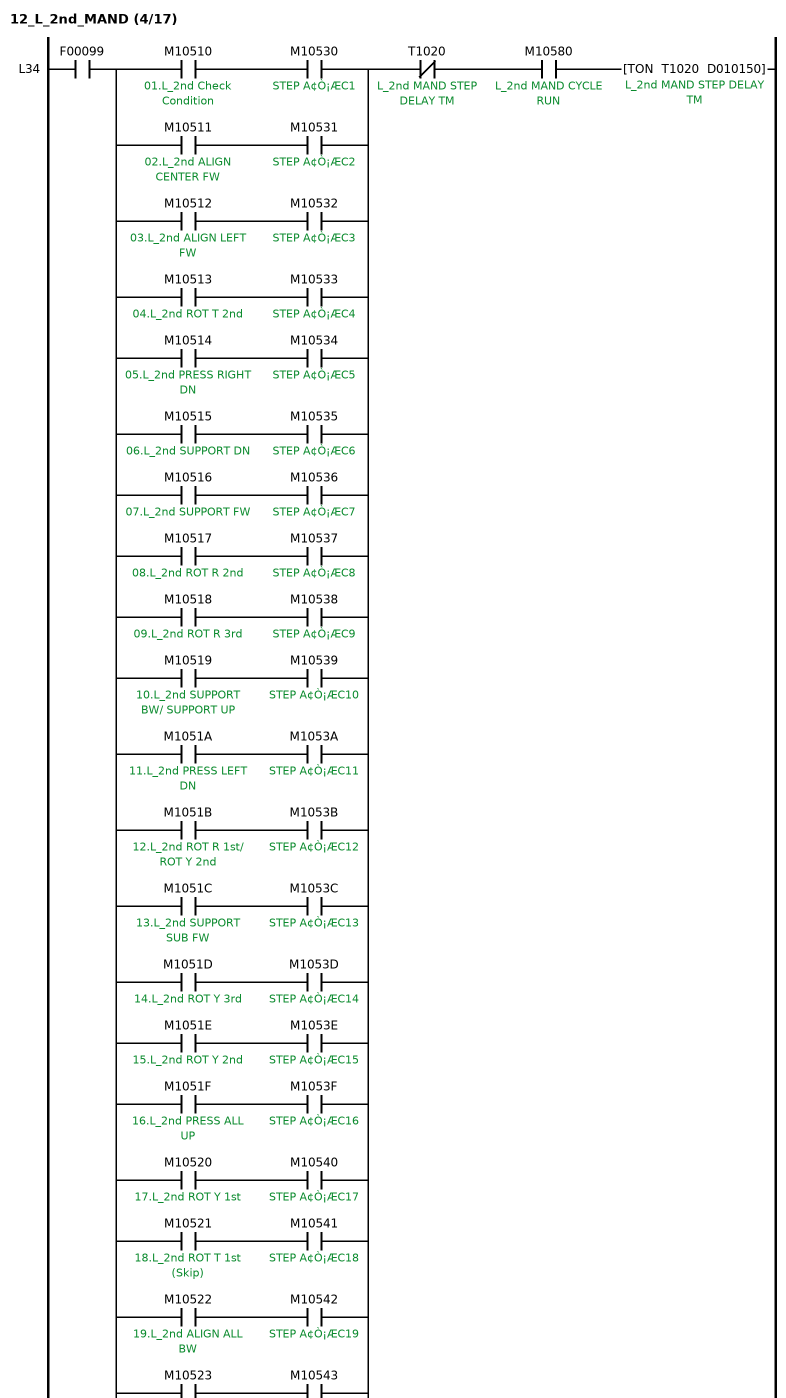
[picture p72: 12_L_2nd_MAND rungs L34-L34]

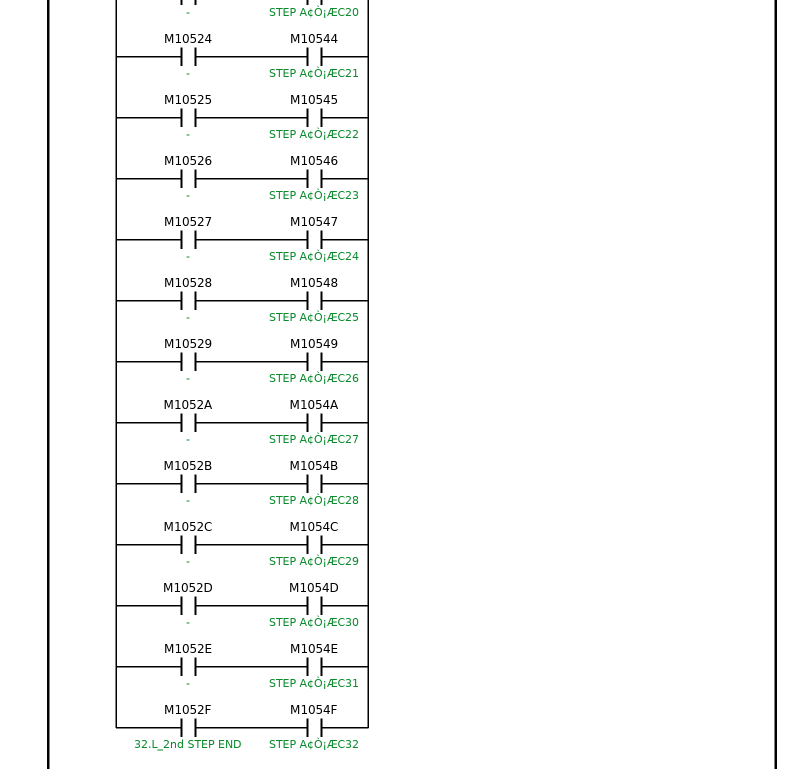
; L34
LOAD      F00099
LOAD      M10510	// 01.L_2nd Check Condition
AND       M10530	// STEP A¢Ò¡ÆC1
LOAD      M10511	// 02.L_2nd ALIGN CENTER FW
AND       M10531	// STEP A¢Ò¡ÆC2
OR LOAD
LOAD      M10512	// 03.L_2nd ALIGN LEFT FW
AND       M10532	// STEP A¢Ò¡ÆC3
OR LOAD
LOAD      M10513	// 04.L_2nd ROT T 2nd
AND       M10533	// STEP A¢Ò¡ÆC4
OR LOAD
LOAD      M10514	// 05.L_2nd PRESS RIGHT DN
AND       M10534	// STEP A¢Ò¡ÆC5
OR LOAD
LOAD      M10515	// 06.L_2nd SUPPORT DN
AND       M10535	// STEP A¢Ò¡ÆC6
OR LOAD
LOAD      M10516	// 07.L_2nd SUPPORT FW
AND       M10536	// STEP A¢Ò¡ÆC7
OR LOAD
LOAD      M10517	// 08.L_2nd ROT R 2nd
AND       M10537	// STEP A¢Ò¡ÆC8
OR LOAD
LOAD      M10518	// 09.L_2nd ROT R 3rd
AND       M10538	// STEP A¢Ò¡ÆC9
OR LOAD
LOAD      M10519	// 10.L_2nd SUPPORT BW/ SUPPORT UP
AND       M10539	// STEP A¢Ò¡ÆC10
OR LOAD
LOAD      M1051A	// 11.L_2nd PRESS LEFT DN
AND       M1053A	// STEP A¢Ò¡ÆC11
OR LOAD
LOAD      M1051B	// 12.L_2nd ROT R 1st/ ROT Y 2nd
AND       M1053B	// STEP A¢Ò¡ÆC12
OR LOAD
LOAD      M1051C	// 13.L_2nd SUPPORT SUB FW
AND       M1053C	// STEP A¢Ò¡ÆC13
OR LOAD
LOAD      M1051D	// 14.L_2nd ROT Y 3rd
AND       M1053D	// STEP A¢Ò¡ÆC14
OR LOAD
LOAD      M1051E	// 15.L_2nd ROT Y 2nd
AND       M1053E	// STEP A¢Ò¡ÆC15
OR LOAD
LOAD      M1051F	// 16.L_2nd PRESS ALL UP
AND       M1053F	// STEP A¢Ò¡ÆC16
OR LOAD
LOAD      M10520	// 17.L_2nd ROT Y 1st
AND       M10540	// STEP A¢Ò¡ÆC17
OR LOAD
LOAD      M10521	// 18.L_2nd ROT T 1st (Skip)
AND       M10541	// STEP A¢Ò¡ÆC18
OR LOAD
LOAD      M10522	// 19.L_2nd ALIGN ALL BW
AND       M10542	// STEP A¢Ò¡ÆC19
OR LOAD
LOAD      M10523	// -
AND       M10543	// STEP A¢Ò¡ÆC20
OR LOAD
LOAD      M10524	// -
AND       M10544	// STEP A¢Ò¡ÆC21
OR LOAD
LOAD      M10525	// -
AND       M10545	// STEP A¢Ò¡ÆC22
OR LOAD
LOAD      M10526	// -
AND       M10546	// STEP A¢Ò¡ÆC23
OR LOAD
LOAD      M10527	// -
AND       M10547	// STEP A¢Ò¡ÆC24
OR LOAD
LOAD      M10528	// -
AND       M10548	// STEP A¢Ò¡ÆC25
OR LOAD
LOAD      M10529	// -
AND       M10549	// STEP A¢Ò¡ÆC26
OR LOAD
LOAD      M1052A	// -
AND       M1054A	// STEP A¢Ò¡ÆC27
OR LOAD
LOAD      M1052B	// -
AND       M1054B	// STEP A¢Ò¡ÆC28
OR LOAD
LOAD      M1052C	// -
AND       M1054C	// STEP A¢Ò¡ÆC29
OR LOAD
LOAD      M1052D	// -
AND       M1054D	// STEP A¢Ò¡ÆC30
OR LOAD
LOAD      M1052E	// -
AND       M1054E	// STEP A¢Ò¡ÆC31
OR LOAD
LOAD      M1052F	// 32.L_2nd STEP END
AND       M1054F	// STEP A¢Ò¡ÆC32
OR LOAD
AND LOAD
AND NOT   T1020	// L_2nd MAND STEP DELAY TM
AND       M10580	// L_2nd MAND CYCLE RUN
TON       T1020 D010150	// L_2nd MAND STEP DELAY TM

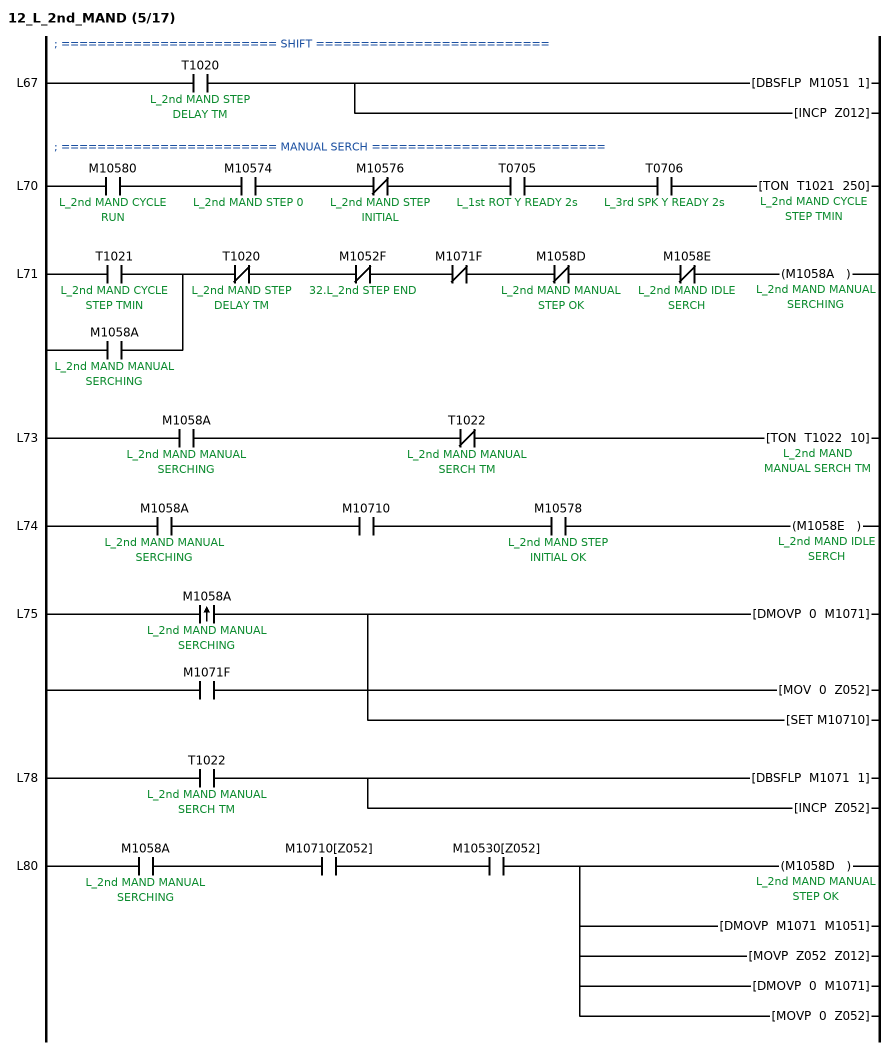
// ======================== SHIFT ==========================
; L67
LOAD      T1020	// L_2nd MAND STEP DELAY TM
DBSFLP    M1051 1
INCP      Z012
// ======================== MANUAL SERCH ==========================
; L70
LOAD      M10580	// L_2nd MAND CYCLE RUN
AND       M10574	// L_2nd MAND STEP 0
AND NOT   M10576	// L_2nd MAND STEP INITIAL
AND       T0705	// L_1st ROT Y READY 2s
AND       T0706	// L_3rd SPK Y READY 2s
TON       T1021 250	// L_2nd MAND CYCLE STEP TMIN
; L71
LOAD      T1021	// L_2nd MAND CYCLE STEP TMIN
OR        M1058A	// L_2nd MAND MANUAL SERCHING
AND NOT   T1020	// L_2nd MAND STEP DELAY TM
AND NOT   M1052F	// 32.L_2nd STEP END
AND NOT   M1071F
AND NOT   M1058D	// L_2nd MAND MANUAL STEP OK
AND NOT   M1058E	// L_2nd MAND IDLE SERCH
OUT       M1058A	// L_2nd MAND MANUAL SERCHING
; L73
LOAD      M1058A	// L_2nd MAND MANUAL SERCHING
AND NOT   T1022	// L_2nd MAND MANUAL SERCH TM
TON       T1022 10	// L_2nd MAND MANUAL SERCH TM
; L74
LOAD      M1058A	// L_2nd MAND MANUAL SERCHING
AND       M10710
AND       M10578	// L_2nd MAND STEP INITIAL OK
OUT       M1058E	// L_2nd MAND IDLE SERCH
; L75
LOADP     M1058A	// L_2nd MAND MANUAL SERCHING
OR        M1071F
DMOVP     0 M1071
MOV       0 Z052
SET       M10710
; L78
LOAD      T1022	// L_2nd MAND MANUAL SERCH TM
DBSFLP    M1071 1
INCP      Z052
; L80
LOAD      M1058A	// L_2nd MAND MANUAL SERCHING
AND       M10710[Z052]
AND       M10530[Z052]
OUT       M1058D	// L_2nd MAND MANUAL STEP OK
DMOVP     M1071 M1051
MOVP      Z052 Z012
DMOVP     0 M1071
MOVP      0 Z052

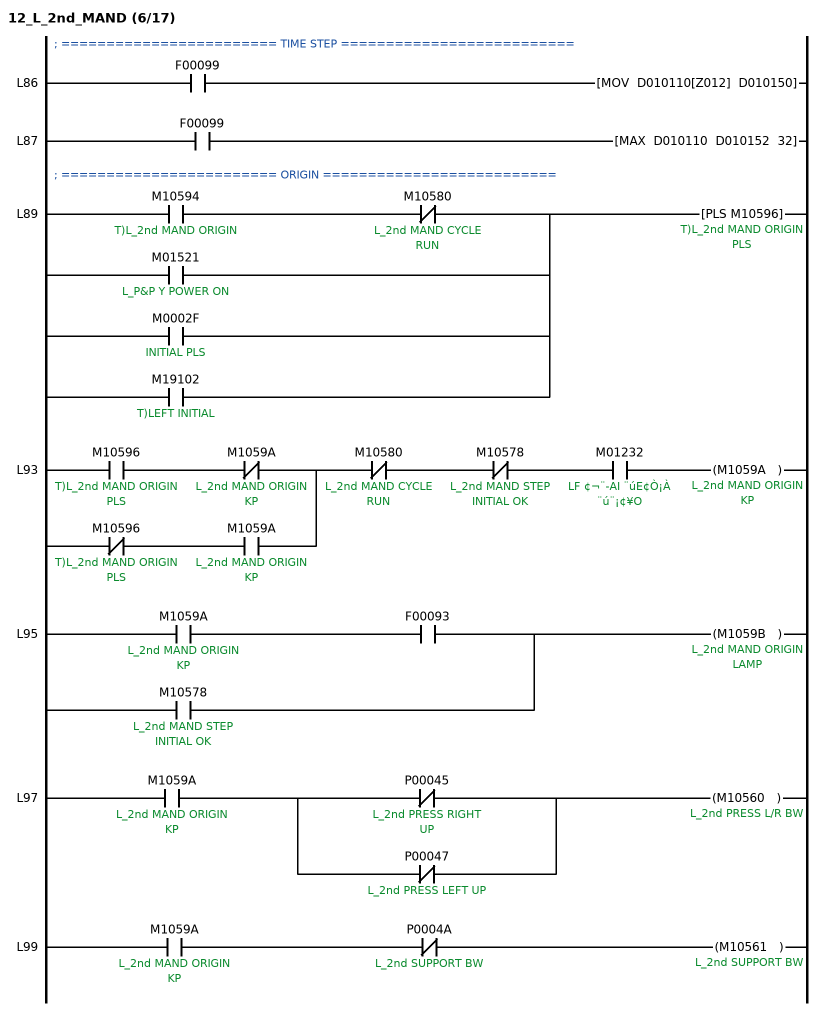
// ======================== TIME STEP ==========================
; L86
LOAD      F00099
MOV       D010110[Z012] D010150
; L87
LOAD      F00099
MAX       D010110 D010152 32
// ======================== ORIGIN ==========================
; L89
LOAD      M10594	// T)L_2nd MAND ORIGIN
AND NOT   M10580	// L_2nd MAND CYCLE RUN
OR        M01521	// L_P&P Y POWER ON
OR        M0002F	// INITIAL PLS
OR        M19102	// T)LEFT INITIAL
OUTP      M10596	// T)L_2nd MAND ORIGIN PLS
; L93
LOAD      M10596	// T)L_2nd MAND ORIGIN PLS
AND NOT   M1059A	// L_2nd MAND ORIGIN KP
LOAD NOT  M10596	// T)L_2nd MAND ORIGIN PLS
AND       M1059A	// L_2nd MAND ORIGIN KP
OR LOAD
AND NOT   M10580	// L_2nd MAND CYCLE RUN
AND NOT   M10578	// L_2nd MAND STEP INITIAL OK
AND       M01232	// LF ¢¬¨­AI ¨úE¢Ò¡À ¨ú¨¡¢¥O
OUT       M1059A	// L_2nd MAND ORIGIN KP
; L95
LOAD      M1059A	// L_2nd MAND ORIGIN KP
AND       F00093
OR        M10578	// L_2nd MAND STEP INITIAL OK
OUT       M1059B	// L_2nd MAND ORIGIN LAMP
; L97
LOAD      M1059A	// L_2nd MAND ORIGIN KP
LOAD NOT  P00045	// L_2nd PRESS RIGHT UP
OR NOT    P00047	// L_2nd PRESS LEFT UP
AND LOAD
OUT       M10560	// L_2nd PRESS L/R BW
; L99
LOAD      M1059A	// L_2nd MAND ORIGIN KP
AND NOT   P0004A	// L_2nd SUPPORT BW
OUT       M10561	// L_2nd SUPPORT BW

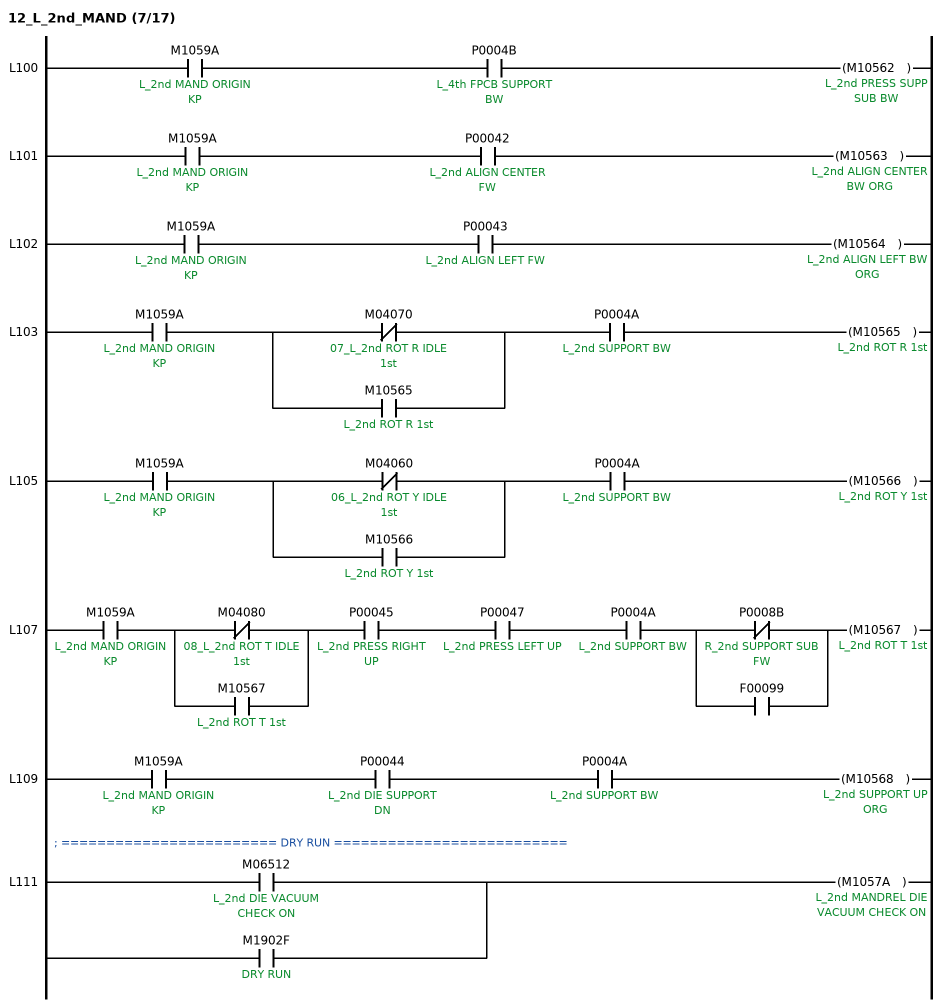
; L100
LOAD      M1059A	// L_2nd MAND ORIGIN KP
AND       P0004B	// L_4th FPCB SUPPORT BW
OUT       M10562	// L_2nd PRESS SUPP SUB BW
; L101
LOAD      M1059A	// L_2nd MAND ORIGIN KP
AND       P00042	// L_2nd ALIGN CENTER FW
OUT       M10563	// L_2nd ALIGN CENTER BW ORG
; L102
LOAD      M1059A	// L_2nd MAND ORIGIN KP
AND       P00043	// L_2nd ALIGN LEFT FW
OUT       M10564	// L_2nd ALIGN LEFT BW ORG
; L103
LOAD      M1059A	// L_2nd MAND ORIGIN KP
LOAD NOT  M04070	// 07_L_2nd ROT R IDLE 1st
OR        M10565	// L_2nd ROT R 1st
AND LOAD
AND       P0004A	// L_2nd SUPPORT BW
OUT       M10565	// L_2nd ROT R 1st
; L105
LOAD      M1059A	// L_2nd MAND ORIGIN KP
LOAD NOT  M04060	// 06_L_2nd ROT Y IDLE 1st
OR        M10566	// L_2nd ROT Y 1st
AND LOAD
AND       P0004A	// L_2nd SUPPORT BW
OUT       M10566	// L_2nd ROT Y 1st
; L107
LOAD      M1059A	// L_2nd MAND ORIGIN KP
LOAD NOT  M04080	// 08_L_2nd ROT T IDLE 1st
OR        M10567	// L_2nd ROT T 1st
AND LOAD
AND       P00045	// L_2nd PRESS RIGHT UP
AND       P00047	// L_2nd PRESS LEFT UP
AND       P0004A	// L_2nd SUPPORT BW
LOAD NOT  P0008B	// R_2nd SUPPORT SUB FW
OR        F00099
AND LOAD
OUT       M10567	// L_2nd ROT T 1st
; L109
LOAD      M1059A	// L_2nd MAND ORIGIN KP
AND       P00044	// L_2nd DIE SUPPORT DN
AND       P0004A	// L_2nd SUPPORT BW
OUT       M10568	// L_2nd SUPPORT UP ORG
// ======================== DRY RUN ==========================
; L111
LOAD      M06512	// L_2nd DIE VACUUM CHECK ON
OR        M1902F	// DRY RUN
OUT       M1057A	// L_2nd MANDREL DIE VACUUM CHECK ON

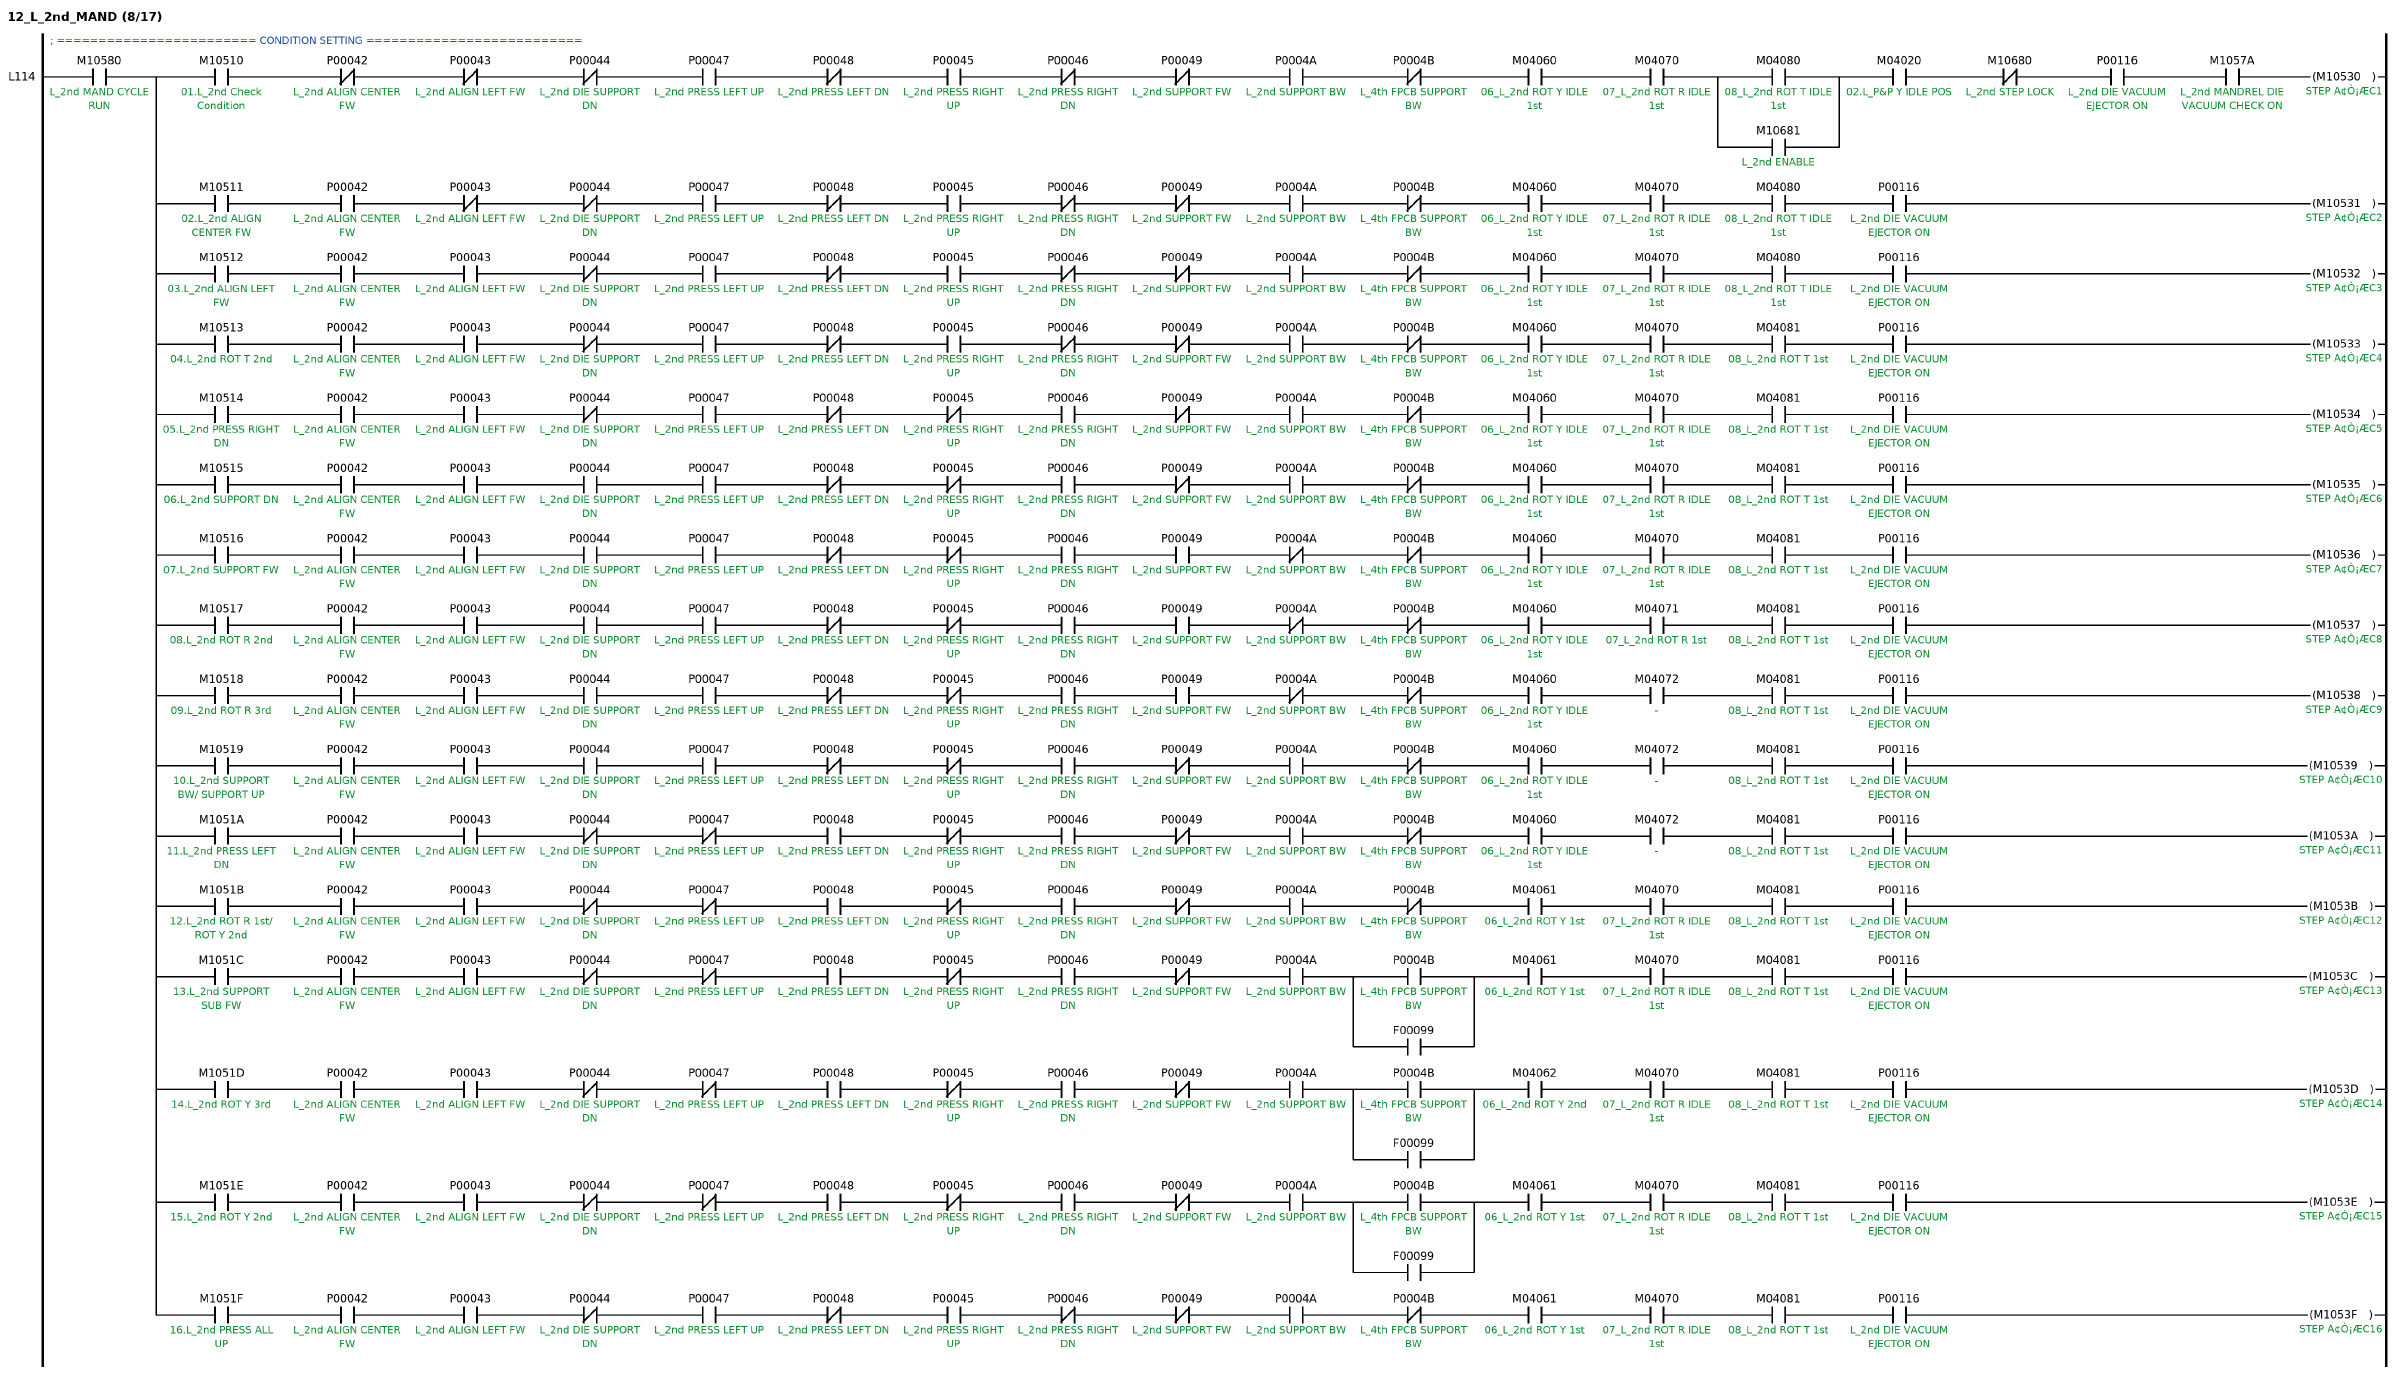
// ======================== CONDITION SETTING ==========================
; L114
LOAD      M10580	// L_2nd MAND CYCLE RUN
MPUSH
AND       M10510	// 01.L_2nd Check Condition
AND NOT   P00042	// L_2nd ALIGN CENTER FW
AND NOT   P00043	// L_2nd ALIGN LEFT FW
AND NOT   P00044	// L_2nd DIE SUPPORT DN
AND       P00047	// L_2nd PRESS LEFT UP
AND NOT   P00048	// L_2nd PRESS LEFT DN
AND       P00045	// L_2nd PRESS RIGHT UP
AND NOT   P00046	// L_2nd PRESS RIGHT DN
AND NOT   P00049	// L_2nd SUPPORT FW
AND       P0004A	// L_2nd SUPPORT BW
AND NOT   P0004B	// L_4th FPCB SUPPORT BW
AND       M04060	// 06_L_2nd ROT Y IDLE 1st
AND       M04070	// 07_L_2nd ROT R IDLE 1st
LOAD      M04080	// 08_L_2nd ROT T IDLE 1st
OR        M10681	// L_2nd ENABLE
AND LOAD
AND       M04020	// 02.L_P&P Y IDLE POS
AND NOT   M10680	// L_2nd STEP LOCK
AND       P00116	// L_2nd DIE VACUUM EJECTOR ON
AND       M1057A	// L_2nd MANDREL DIE VACUUM CHECK ON
OUT       M10530	// STEP A¢Ò¡ÆC1
MLOAD
AND       M10511	// 02.L_2nd ALIGN CENTER FW
AND       P00042	// L_2nd ALIGN CENTER FW
AND NOT   P00043	// L_2nd ALIGN LEFT FW
AND NOT   P00044	// L_2nd DIE SUPPORT DN
AND       P00047	// L_2nd PRESS LEFT UP
AND NOT   P00048	// L_2nd PRESS LEFT DN
AND       P00045	// L_2nd PRESS RIGHT UP
AND NOT   P00046	// L_2nd PRESS RIGHT DN
AND NOT   P00049	// L_2nd SUPPORT FW
AND       P0004A	// L_2nd SUPPORT BW
AND NOT   P0004B	// L_4th FPCB SUPPORT BW
AND       M04060	// 06_L_2nd ROT Y IDLE 1st
AND       M04070	// 07_L_2nd ROT R IDLE 1st
AND       M04080	// 08_L_2nd ROT T IDLE 1st
AND       P00116	// L_2nd DIE VACUUM EJECTOR ON
OUT       M10531	// STEP A¢Ò¡ÆC2
MLOAD
AND       M10512	// 03.L_2nd ALIGN LEFT FW
AND       P00042	// L_2nd ALIGN CENTER FW
AND       P00043	// L_2nd ALIGN LEFT FW
AND NOT   P00044	// L_2nd DIE SUPPORT DN
AND       P00047	// L_2nd PRESS LEFT UP
AND NOT   P00048	// L_2nd PRESS LEFT DN
AND       P00045	// L_2nd PRESS RIGHT UP
AND NOT   P00046	// L_2nd PRESS RIGHT DN
AND NOT   P00049	// L_2nd SUPPORT FW
AND       P0004A	// L_2nd SUPPORT BW
AND NOT   P0004B	// L_4th FPCB SUPPORT BW
AND       M04060	// 06_L_2nd ROT Y IDLE 1st
AND       M04070	// 07_L_2nd ROT R IDLE 1st
AND       M04080	// 08_L_2nd ROT T IDLE 1st
AND       P00116	// L_2nd DIE VACUUM EJECTOR ON
OUT       M10532	// STEP A¢Ò¡ÆC3
MLOAD
AND       M10513	// 04.L_2nd ROT T 2nd
AND       P00042	// L_2nd ALIGN CENTER FW
AND       P00043	// L_2nd ALIGN LEFT FW
AND NOT   P00044	// L_2nd DIE SUPPORT DN
AND       P00047	// L_2nd PRESS LEFT UP
AND NOT   P00048	// L_2nd PRESS LEFT DN
AND       P00045	// L_2nd PRESS RIGHT UP
AND NOT   P00046	// L_2nd PRESS RIGHT DN
AND NOT   P00049	// L_2nd SUPPORT FW
AND       P0004A	// L_2nd SUPPORT BW
AND NOT   P0004B	// L_4th FPCB SUPPORT BW
AND       M04060	// 06_L_2nd ROT Y IDLE 1st
AND       M04070	// 07_L_2nd ROT R IDLE 1st
AND       M04081	// 08_L_2nd ROT T 1st
AND       P00116	// L_2nd DIE VACUUM EJECTOR ON
OUT       M10533	// STEP A¢Ò¡ÆC4
MLOAD
AND       M10514	// 05.L_2nd PRESS RIGHT DN
AND       P00042	// L_2nd ALIGN CENTER FW
AND       P00043	// L_2nd ALIGN LEFT FW
AND NOT   P00044	// L_2nd DIE SUPPORT DN
AND       P00047	// L_2nd PRESS LEFT UP
AND NOT   P00048	// L_2nd PRESS LEFT DN
AND NOT   P00045	// L_2nd PRESS RIGHT UP
AND       P00046	// L_2nd PRESS RIGHT DN
AND NOT   P00049	// L_2nd SUPPORT FW
AND       P0004A	// L_2nd SUPPORT BW
AND NOT   P0004B	// L_4th FPCB SUPPORT BW
AND       M04060	// 06_L_2nd ROT Y IDLE 1st
AND       M04070	// 07_L_2nd ROT R IDLE 1st
AND       M04081	// 08_L_2nd ROT T 1st
AND       P00116	// L_2nd DIE VACUUM EJECTOR ON
OUT       M10534	// STEP A¢Ò¡ÆC5
MLOAD
AND       M10515	// 06.L_2nd SUPPORT DN
AND       P00042	// L_2nd ALIGN CENTER FW
AND       P00043	// L_2nd ALIGN LEFT FW
AND       P00044	// L_2nd DIE SUPPORT DN
AND       P00047	// L_2nd PRESS LEFT UP
AND NOT   P00048	// L_2nd PRESS LEFT DN
AND NOT   P00045	// L_2nd PRESS RIGHT UP
AND       P00046	// L_2nd PRESS RIGHT DN
AND NOT   P00049	// L_2nd SUPPORT FW
AND       P0004A	// L_2nd SUPPORT BW
AND NOT   P0004B	// L_4th FPCB SUPPORT BW
AND       M04060	// 06_L_2nd ROT Y IDLE 1st
AND       M04070	// 07_L_2nd ROT R IDLE 1st
AND       M04081	// 08_L_2nd ROT T 1st
AND       P00116	// L_2nd DIE VACUUM EJECTOR ON
OUT       M10535	// STEP A¢Ò¡ÆC6
MLOAD
AND       M10516	// 07.L_2nd SUPPORT FW
AND       P00042	// L_2nd ALIGN CENTER FW
AND       P00043	// L_2nd ALIGN LEFT FW
AND       P00044	// L_2nd DIE SUPPORT DN
AND       P00047	// L_2nd PRESS LEFT UP
AND NOT   P00048	// L_2nd PRESS LEFT DN
AND NOT   P00045	// L_2nd PRESS RIGHT UP
AND       P00046	// L_2nd PRESS RIGHT DN
AND       P00049	// L_2nd SUPPORT FW
AND NOT   P0004A	// L_2nd SUPPORT BW
AND NOT   P0004B	// L_4th FPCB SUPPORT BW
AND       M04060	// 06_L_2nd ROT Y IDLE 1st
AND       M04070	// 07_L_2nd ROT R IDLE 1st
AND       M04081	// 08_L_2nd ROT T 1st
AND       P00116	// L_2nd DIE VACUUM EJECTOR ON
OUT       M10536	// STEP A¢Ò¡ÆC7
MLOAD
AND       M10517	// 08.L_2nd ROT R 2nd
AND       P00042	// L_2nd ALIGN CENTER FW
AND       P00043	// L_2nd ALIGN LEFT FW
AND       P00044	// L_2nd DIE SUPPORT DN
AND       P00047	// L_2nd PRESS LEFT UP
AND NOT   P00048	// L_2nd PRESS LEFT DN
AND NOT   P00045	// L_2nd PRESS RIGHT UP
AND       P00046	// L_2nd PRESS RIGHT DN
AND       P00049	// L_2nd SUPPORT FW
AND NOT   P0004A	// L_2nd SUPPORT BW
AND NOT   P0004B	// L_4th FPCB SUPPORT BW
AND       M04060	// 06_L_2nd ROT Y IDLE 1st
AND       M04071	// 07_L_2nd ROT R 1st
AND       M04081	// 08_L_2nd ROT T 1st
AND       P00116	// L_2nd DIE VACUUM EJECTOR ON
OUT       M10537	// STEP A¢Ò¡ÆC8
MLOAD
AND       M10518	// 09.L_2nd ROT R 3rd
AND       P00042	// L_2nd ALIGN CENTER FW
AND       P00043	// L_2nd ALIGN LEFT FW
AND       P00044	// L_2nd DIE SUPPORT DN
AND       P00047	// L_2nd PRESS LEFT UP
AND NOT   P00048	// L_2nd PRESS LEFT DN
AND NOT   P00045	// L_2nd PRESS RIGHT UP
AND       P00046	// L_2nd PRESS RIGHT DN
AND       P00049	// L_2nd SUPPORT FW
AND NOT   P0004A	// L_2nd SUPPORT BW
AND NOT   P0004B	// L_4th FPCB SUPPORT BW
AND       M04060	// 06_L_2nd ROT Y IDLE 1st
AND       M04072	// -
AND       M04081	// 08_L_2nd ROT T 1st
AND       P00116	// L_2nd DIE VACUUM EJECTOR ON
OUT       M10538	// STEP A¢Ò¡ÆC9
MLOAD
AND       M10519	// 10.L_2nd SUPPORT BW/ SUPPORT UP
AND       P00042	// L_2nd ALIGN CENTER FW
AND       P00043	// L_2nd ALIGN LEFT FW
AND       P00044	// L_2nd DIE SUPPORT DN
AND       P00047	// L_2nd PRESS LEFT UP
AND NOT   P00048	// L_2nd PRESS LEFT DN
AND NOT   P00045	// L_2nd PRESS RIGHT UP
AND       P00046	// L_2nd PRESS RIGHT DN
AND NOT   P00049	// L_2nd SUPPORT FW
AND       P0004A	// L_2nd SUPPORT BW
AND NOT   P0004B	// L_4th FPCB SUPPORT BW
AND       M04060	// 06_L_2nd ROT Y IDLE 1st
AND       M04072	// -
AND       M04081	// 08_L_2nd ROT T 1st
AND       P00116	// L_2nd DIE VACUUM EJECTOR ON
OUT       M10539	// STEP A¢Ò¡ÆC10
MLOAD
AND       M1051A	// 11.L_2nd PRESS LEFT DN
AND       P00042	// L_2nd ALIGN CENTER FW
AND       P00043	// L_2nd ALIGN LEFT FW
AND NOT   P00044	// L_2nd DIE SUPPORT DN
AND NOT   P00047	// L_2nd PRESS LEFT UP
AND       P00048	// L_2nd PRESS LEFT DN
AND NOT   P00045	// L_2nd PRESS RIGHT UP
AND       P00046	// L_2nd PRESS RIGHT DN
AND NOT   P00049	// L_2nd SUPPORT FW
AND       P0004A	// L_2nd SUPPORT BW
AND NOT   P0004B	// L_4th FPCB SUPPORT BW
AND       M04060	// 06_L_2nd ROT Y IDLE 1st
AND       M04072	// -
AND       M04081	// 08_L_2nd ROT T 1st
AND       P00116	// L_2nd DIE VACUUM EJECTOR ON
OUT       M1053A	// STEP A¢Ò¡ÆC11
MLOAD
AND       M1051B	// 12.L_2nd ROT R 1st/ ROT Y 2nd
AND       P00042	// L_2nd ALIGN CENTER FW
AND       P00043	// L_2nd ALIGN LEFT FW
AND NOT   P00044	// L_2nd DIE SUPPORT DN
AND NOT   P00047	// L_2nd PRESS LEFT UP
AND       P00048	// L_2nd PRESS LEFT DN
AND NOT   P00045	// L_2nd PRESS RIGHT UP
AND       P00046	// L_2nd PRESS RIGHT DN
AND NOT   P00049	// L_2nd SUPPORT FW
AND       P0004A	// L_2nd SUPPORT BW
AND NOT   P0004B	// L_4th FPCB SUPPORT BW
AND       M04061	// 06_L_2nd ROT Y 1st
AND       M04070	// 07_L_2nd ROT R IDLE 1st
AND       M04081	// 08_L_2nd ROT T 1st
AND       P00116	// L_2nd DIE VACUUM EJECTOR ON
OUT       M1053B	// STEP A¢Ò¡ÆC12
MLOAD
AND       M1051C	// 13.L_2nd SUPPORT SUB FW
AND       P00042	// L_2nd ALIGN CENTER FW
AND       P00043	// L_2nd ALIGN LEFT FW
AND NOT   P00044	// L_2nd DIE SUPPORT DN
AND NOT   P00047	// L_2nd PRESS LEFT UP
AND       P00048	// L_2nd PRESS LEFT DN
AND NOT   P00045	// L_2nd PRESS RIGHT UP
AND       P00046	// L_2nd PRESS RIGHT DN
AND NOT   P00049	// L_2nd SUPPORT FW
AND       P0004A	// L_2nd SUPPORT BW
LOAD      P0004B	// L_4th FPCB SUPPORT BW
OR        F00099
AND LOAD
AND       M04061	// 06_L_2nd ROT Y 1st
AND       M04070	// 07_L_2nd ROT R IDLE 1st
AND       M04081	// 08_L_2nd ROT T 1st
AND       P00116	// L_2nd DIE VACUUM EJECTOR ON
OUT       M1053C	// STEP A¢Ò¡ÆC13
MLOAD
AND       M1051D	// 14.L_2nd ROT Y 3rd
AND       P00042	// L_2nd ALIGN CENTER FW
AND       P00043	// L_2nd ALIGN LEFT FW
AND NOT   P00044	// L_2nd DIE SUPPORT DN
AND NOT   P00047	// L_2nd PRESS LEFT UP
AND       P00048	// L_2nd PRESS LEFT DN
AND NOT   P00045	// L_2nd PRESS RIGHT UP
AND       P00046	// L_2nd PRESS RIGHT DN
AND NOT   P00049	// L_2nd SUPPORT FW
AND       P0004A	// L_2nd SUPPORT BW
LOAD      P0004B	// L_4th FPCB SUPPORT BW
OR        F00099
AND LOAD
AND       M04062	// 06_L_2nd ROT Y 2nd
AND       M04070	// 07_L_2nd ROT R IDLE 1st
AND       M04081	// 08_L_2nd ROT T 1st
AND       P00116	// L_2nd DIE VACUUM EJECTOR ON
OUT       M1053D	// STEP A¢Ò¡ÆC14
MLOAD
AND       M1051E	// 15.L_2nd ROT Y 2nd
AND       P00042	// L_2nd ALIGN CENTER FW
AND       P00043	// L_2nd ALIGN LEFT FW
AND NOT   P00044	// L_2nd DIE SUPPORT DN
AND NOT   P00047	// L_2nd PRESS LEFT UP
AND       P00048	// L_2nd PRESS LEFT DN
AND NOT   P00045	// L_2nd PRESS RIGHT UP
AND       P00046	// L_2nd PRESS RIGHT DN
AND NOT   P00049	// L_2nd SUPPORT FW
AND       P0004A	// L_2nd SUPPORT BW
LOAD      P0004B	// L_4th FPCB SUPPORT BW
OR        F00099
AND LOAD
AND       M04061	// 06_L_2nd ROT Y 1st
AND       M04070	// 07_L_2nd ROT R IDLE 1st
AND       M04081	// 08_L_2nd ROT T 1st
AND       P00116	// L_2nd DIE VACUUM EJECTOR ON
OUT       M1053E	// STEP A¢Ò¡ÆC15
MPOP
AND       M1051F	// 16.L_2nd PRESS ALL UP
AND       P00042	// L_2nd ALIGN CENTER FW
AND       P00043	// L_2nd ALIGN LEFT FW
AND NOT   P00044	// L_2nd DIE SUPPORT DN
AND       P00047	// L_2nd PRESS LEFT UP
AND NOT   P00048	// L_2nd PRESS LEFT DN
AND       P00045	// L_2nd PRESS RIGHT UP
AND NOT   P00046	// L_2nd PRESS RIGHT DN
AND NOT   P00049	// L_2nd SUPPORT FW
AND       P0004A	// L_2nd SUPPORT BW
AND NOT   P0004B	// L_4th FPCB SUPPORT BW
AND       M04061	// 06_L_2nd ROT Y 1st
AND       M04070	// 07_L_2nd ROT R IDLE 1st
AND       M04081	// 08_L_2nd ROT T 1st
AND       P00116	// L_2nd DIE VACUUM EJECTOR ON
OUT       M1053F	// STEP A¢Ò¡ÆC16

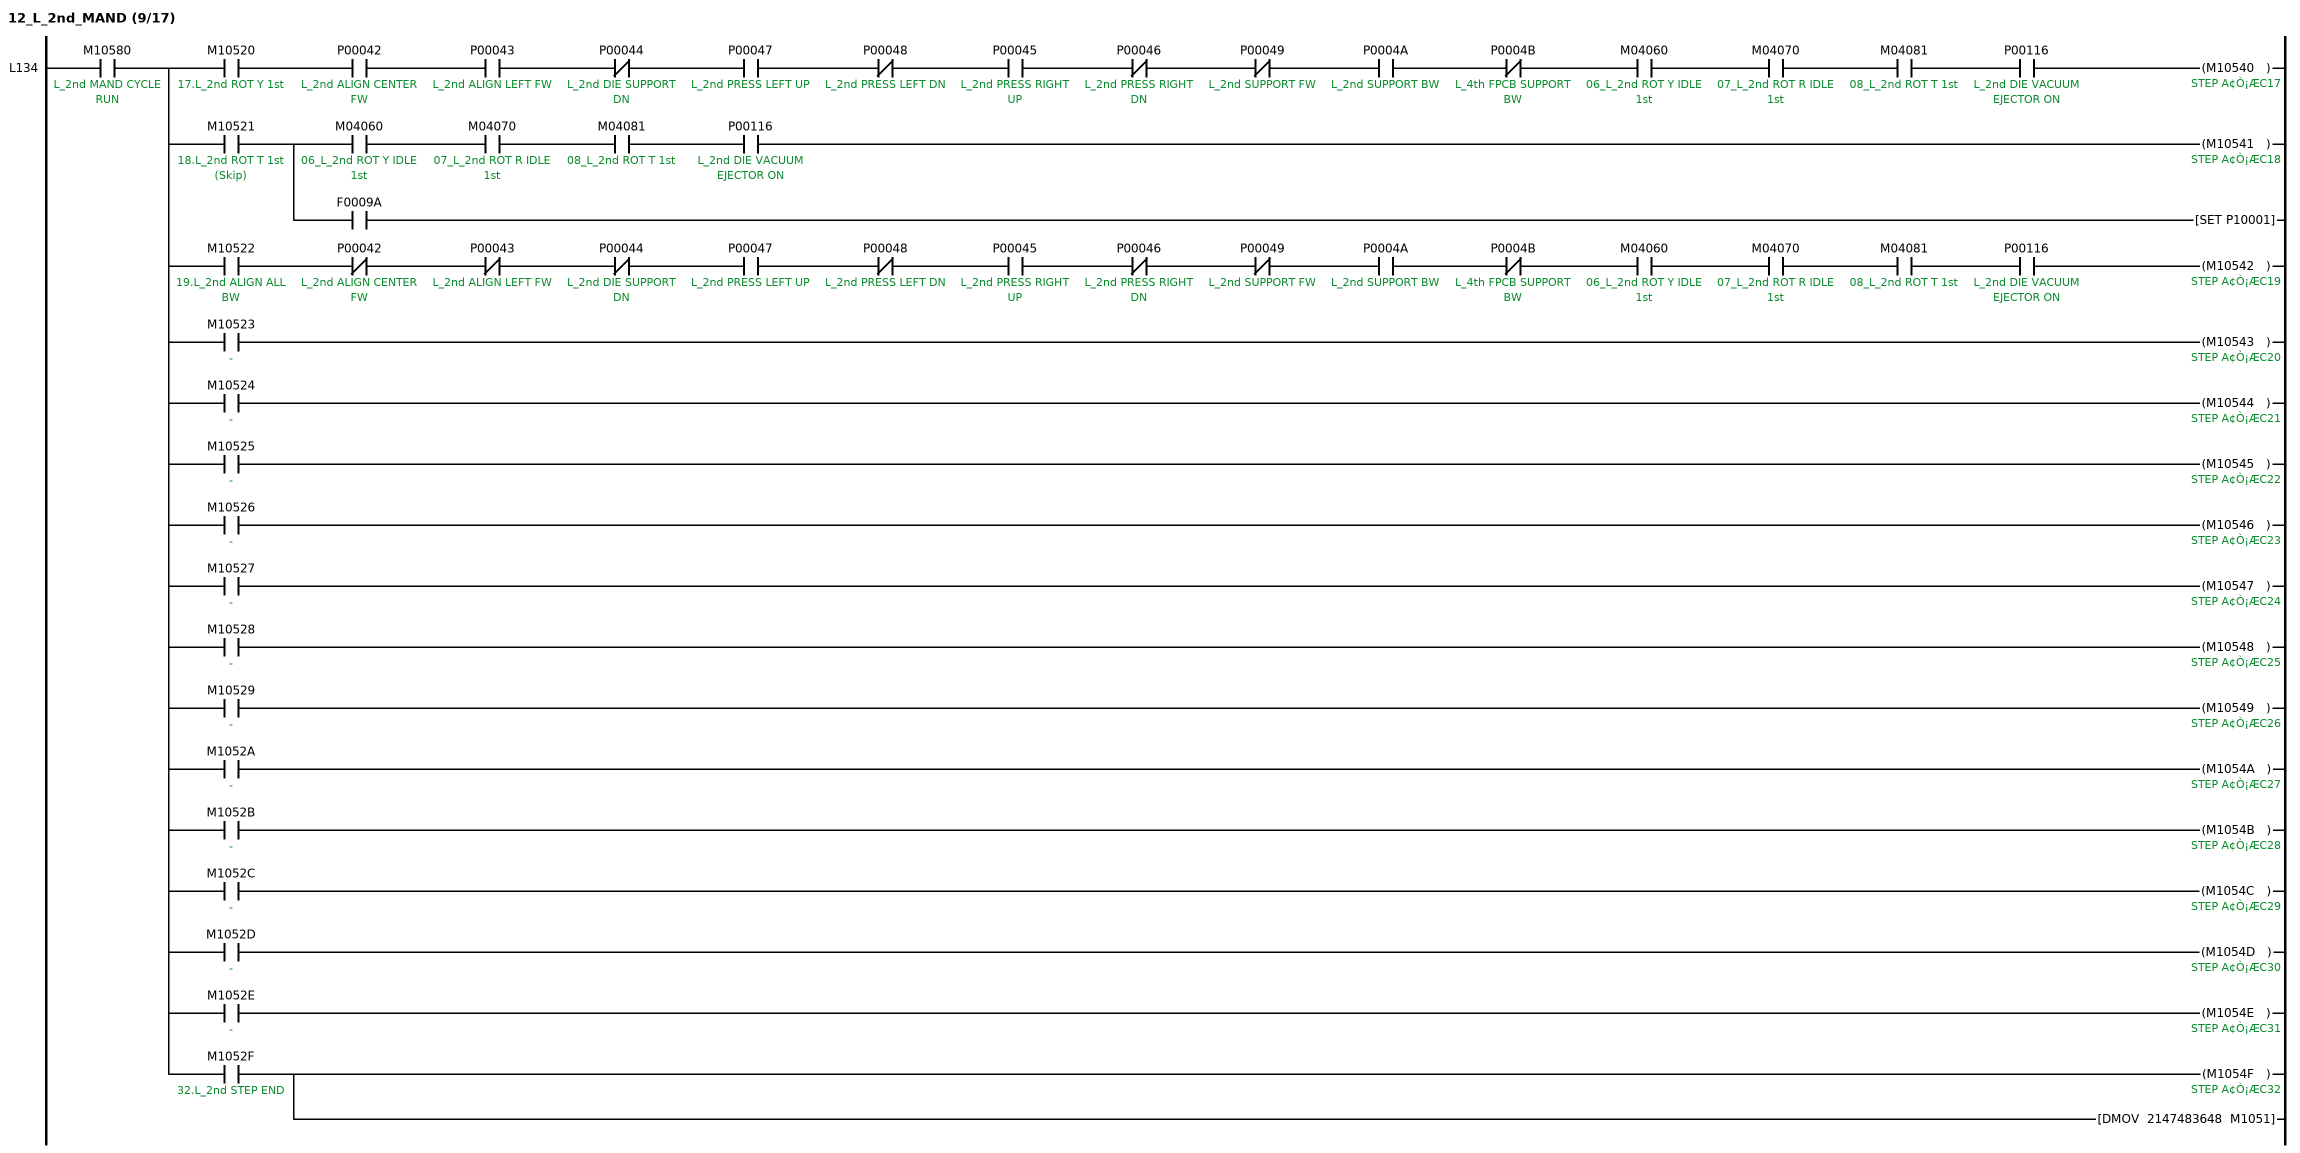
; L134
LOAD      M10580	// L_2nd MAND CYCLE RUN
MPUSH
AND       M10520	// 17.L_2nd ROT Y 1st
AND       P00042	// L_2nd ALIGN CENTER FW
AND       P00043	// L_2nd ALIGN LEFT FW
AND NOT   P00044	// L_2nd DIE SUPPORT DN
AND       P00047	// L_2nd PRESS LEFT UP
AND NOT   P00048	// L_2nd PRESS LEFT DN
AND       P00045	// L_2nd PRESS RIGHT UP
AND NOT   P00046	// L_2nd PRESS RIGHT DN
AND NOT   P00049	// L_2nd SUPPORT FW
AND       P0004A	// L_2nd SUPPORT BW
AND NOT   P0004B	// L_4th FPCB SUPPORT BW
AND       M04060	// 06_L_2nd ROT Y IDLE 1st
AND       M04070	// 07_L_2nd ROT R IDLE 1st
AND       M04081	// 08_L_2nd ROT T 1st
AND       P00116	// L_2nd DIE VACUUM EJECTOR ON
OUT       M10540	// STEP A¢Ò¡ÆC17
MLOAD
AND       M10521	// 18.L_2nd ROT T 1st (Skip)
MPUSH
AND       M04060	// 06_L_2nd ROT Y IDLE 1st
AND       M04070	// 07_L_2nd ROT R IDLE 1st
AND       M04081	// 08_L_2nd ROT T 1st
AND       P00116	// L_2nd DIE VACUUM EJECTOR ON
OUT       M10541	// STEP A¢Ò¡ÆC18
MPOP
AND       F0009A
SET       P10001
MLOAD
AND       M10522	// 19.L_2nd ALIGN ALL BW
AND NOT   P00042	// L_2nd ALIGN CENTER FW
AND NOT   P00043	// L_2nd ALIGN LEFT FW
AND NOT   P00044	// L_2nd DIE SUPPORT DN
AND       P00047	// L_2nd PRESS LEFT UP
AND NOT   P00048	// L_2nd PRESS LEFT DN
AND       P00045	// L_2nd PRESS RIGHT UP
AND NOT   P00046	// L_2nd PRESS RIGHT DN
AND NOT   P00049	// L_2nd SUPPORT FW
AND       P0004A	// L_2nd SUPPORT BW
AND NOT   P0004B	// L_4th FPCB SUPPORT BW
AND       M04060	// 06_L_2nd ROT Y IDLE 1st
AND       M04070	// 07_L_2nd ROT R IDLE 1st
AND       M04081	// 08_L_2nd ROT T 1st
AND       P00116	// L_2nd DIE VACUUM EJECTOR ON
OUT       M10542	// STEP A¢Ò¡ÆC19
MLOAD
AND       M10523	// -
OUT       M10543	// STEP A¢Ò¡ÆC20
MLOAD
AND       M10524	// -
OUT       M10544	// STEP A¢Ò¡ÆC21
MLOAD
AND       M10525	// -
OUT       M10545	// STEP A¢Ò¡ÆC22
MLOAD
AND       M10526	// -
OUT       M10546	// STEP A¢Ò¡ÆC23
MLOAD
AND       M10527	// -
OUT       M10547	// STEP A¢Ò¡ÆC24
MLOAD
AND       M10528	// -
OUT       M10548	// STEP A¢Ò¡ÆC25
MLOAD
AND       M10529	// -
OUT       M10549	// STEP A¢Ò¡ÆC26
MLOAD
AND       M1052A	// -
OUT       M1054A	// STEP A¢Ò¡ÆC27
MLOAD
AND       M1052B	// -
OUT       M1054B	// STEP A¢Ò¡ÆC28
MLOAD
AND       M1052C	// -
OUT       M1054C	// STEP A¢Ò¡ÆC29
MLOAD
AND       M1052D	// -
OUT       M1054D	// STEP A¢Ò¡ÆC30
MLOAD
AND       M1052E	// -
OUT       M1054E	// STEP A¢Ò¡ÆC31
MPOP
AND       M1052F	// 32.L_2nd STEP END
OUT       M1054F	// STEP A¢Ò¡ÆC32
DMOV      2147483648 M1051

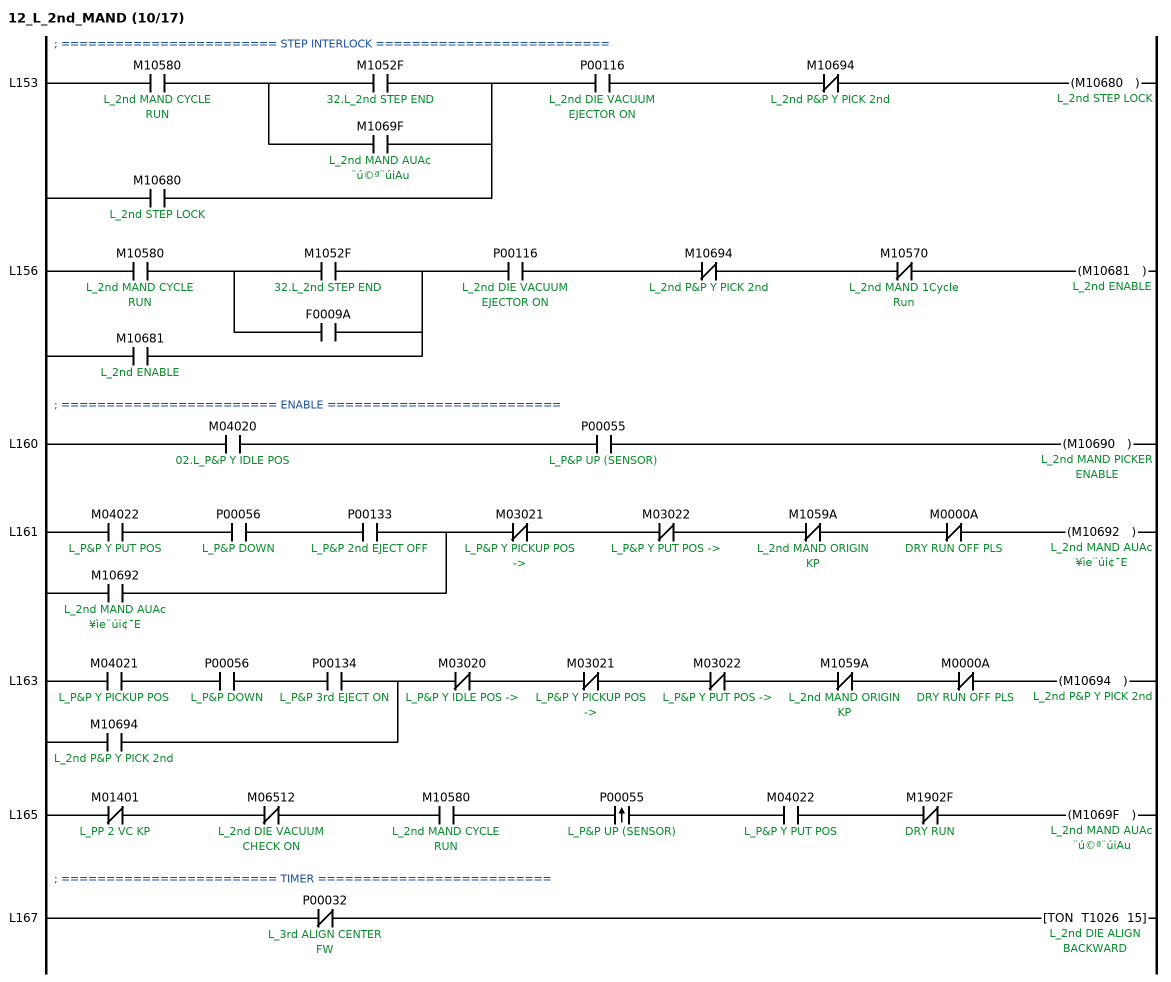
// ======================== STEP INTERLOCK ==========================
; L153
LOAD      M10580	// L_2nd MAND CYCLE RUN
LOAD      M1052F	// 32.L_2nd STEP END
OR        M1069F	// L_2nd MAND AUAc ¨ú©ª¨úiAu
AND LOAD
OR        M10680	// L_2nd STEP LOCK
AND       P00116	// L_2nd DIE VACUUM EJECTOR ON
AND NOT   M10694	// L_2nd P&P Y PICK 2nd
OUT       M10680	// L_2nd STEP LOCK
; L156
LOAD      M10580	// L_2nd MAND CYCLE RUN
LOAD      M1052F	// 32.L_2nd STEP END
OR        F0009A
AND LOAD
OR        M10681	// L_2nd ENABLE
AND       P00116	// L_2nd DIE VACUUM EJECTOR ON
AND NOT   M10694	// L_2nd P&P Y PICK 2nd
AND NOT   M10570	// L_2nd MAND 1Cycle Run
OUT       M10681	// L_2nd ENABLE
// ======================== ENABLE ==========================
; L160
LOAD      M04020	// 02.L_P&P Y IDLE POS
AND       P00055	// L_P&P UP (SENSOR)
OUT       M10690	// L_2nd MAND PICKER ENABLE
; L161
LOAD      M04022	// L_P&P Y PUT POS
AND       P00056	// L_P&P DOWN
AND       P00133	// L_P&P 2nd EJECT OFF
OR        M10692	// L_2nd MAND AUAc ¥ìe¨úi¢¯E
AND NOT   M03021	// L_P&P Y PICKUP POS ->
AND NOT   M03022	// L_P&P Y PUT POS ->
AND NOT   M1059A	// L_2nd MAND ORIGIN KP
AND NOT   M0000A	// DRY RUN OFF PLS
OUT       M10692	// L_2nd MAND AUAc ¥ìe¨úi¢¯E
; L163
LOAD      M04021	// L_P&P Y PICKUP POS
AND       P00056	// L_P&P DOWN
AND       P00134	// L_P&P 3rd EJECT ON
OR        M10694	// L_2nd P&P Y PICK 2nd
AND NOT   M03020	// L_P&P Y IDLE POS ->
AND NOT   M03021	// L_P&P Y PICKUP POS ->
AND NOT   M03022	// L_P&P Y PUT POS ->
AND NOT   M1059A	// L_2nd MAND ORIGIN KP
AND NOT   M0000A	// DRY RUN OFF PLS
OUT       M10694	// L_2nd P&P Y PICK 2nd
; L165
LOAD NOT  M01401	// L_PP 2 VC KP
AND NOT   M06512	// L_2nd DIE VACUUM CHECK ON
AND       M10580	// L_2nd MAND CYCLE RUN
ANDP      P00055	// L_P&P UP (SENSOR)
AND       M04022	// L_P&P Y PUT POS
AND NOT   M1902F	// DRY RUN
OUT       M1069F	// L_2nd MAND AUAc ¨ú©ª¨úiAu
// ======================== TIMER ==========================
; L167
LOAD NOT  P00032	// L_3rd ALIGN CENTER FW
TON       T1026 15	// L_2nd DIE ALIGN BACKWARD

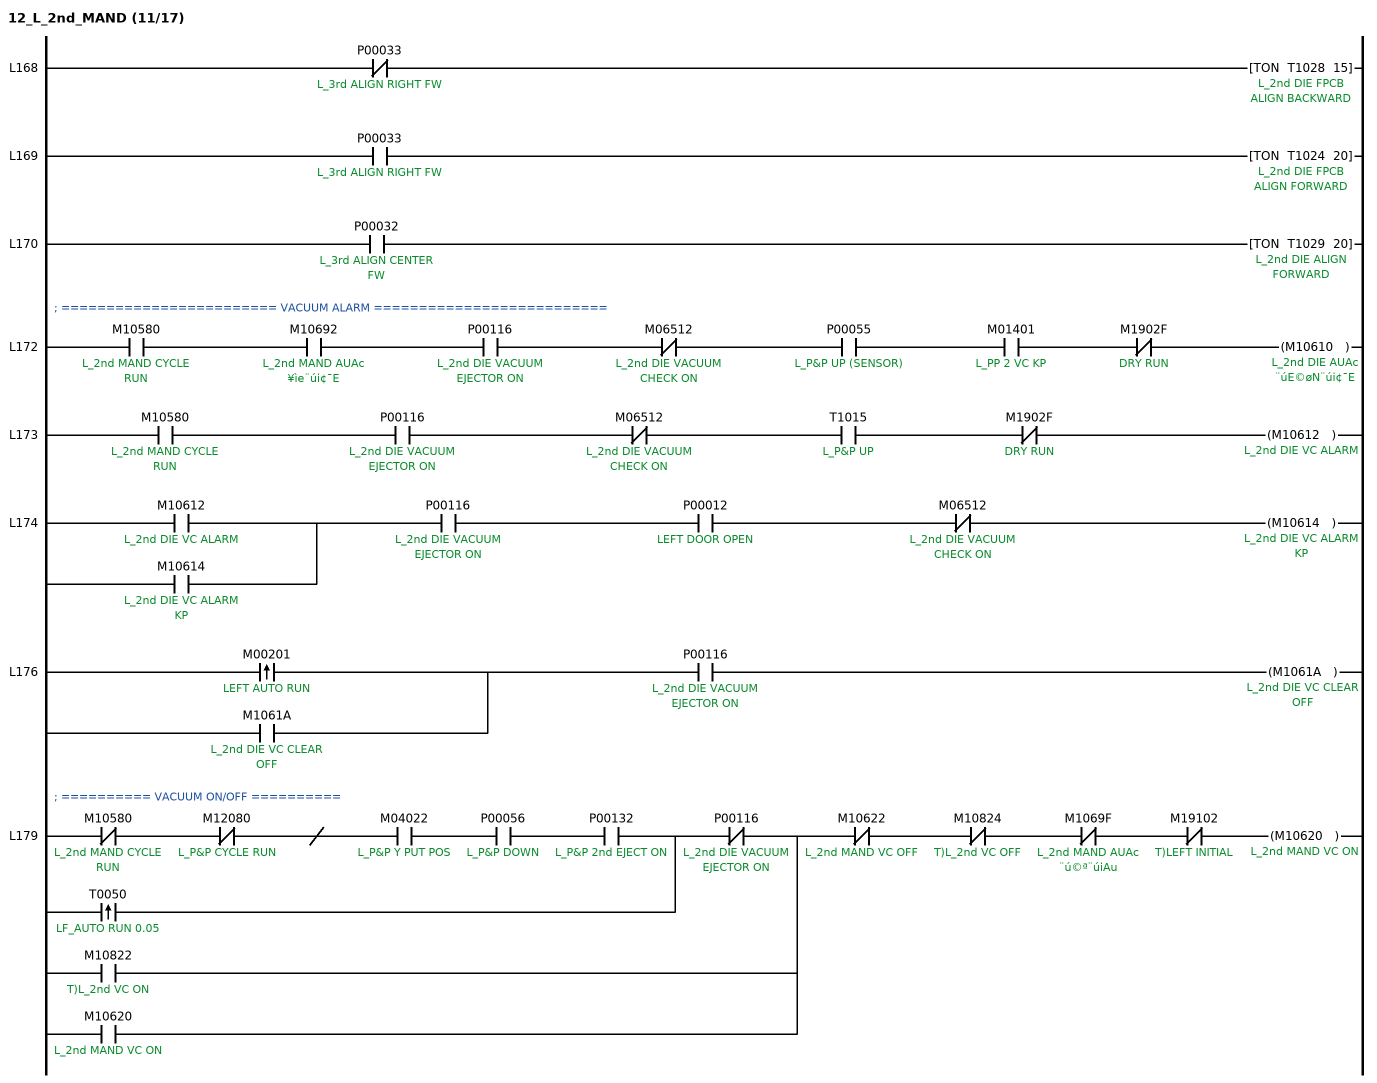
; L168
LOAD NOT  P00033	// L_3rd ALIGN RIGHT FW
TON       T1028 15	// L_2nd DIE FPCB ALIGN BACKWARD
; L169
LOAD      P00033	// L_3rd ALIGN RIGHT FW
TON       T1024 20	// L_2nd DIE FPCB ALIGN FORWARD
; L170
LOAD      P00032	// L_3rd ALIGN CENTER FW
TON       T1029 20	// L_2nd DIE ALIGN FORWARD
// ======================== VACUUM ALARM ==========================
; L172
LOAD      M10580	// L_2nd MAND CYCLE RUN
AND       M10692	// L_2nd MAND AUAc ¥ìe¨úi¢¯E
AND       P00116	// L_2nd DIE VACUUM EJECTOR ON
AND NOT   M06512	// L_2nd DIE VACUUM CHECK ON
AND       P00055	// L_P&P UP (SENSOR)
AND       M01401	// L_PP 2 VC KP
AND NOT   M1902F	// DRY RUN
OUT       M10610	// L_2nd DIE AUAc ¨úE©øN¨úi¢¯E
; L173
LOAD      M10580	// L_2nd MAND CYCLE RUN
AND       P00116	// L_2nd DIE VACUUM EJECTOR ON
AND NOT   M06512	// L_2nd DIE VACUUM CHECK ON
AND       T1015	// L_P&P UP
AND NOT   M1902F	// DRY RUN
OUT       M10612	// L_2nd DIE VC ALARM
; L174
LOAD      M10612	// L_2nd DIE VC ALARM
OR        M10614	// L_2nd DIE VC ALARM KP
AND       P00116	// L_2nd DIE VACUUM EJECTOR ON
AND       P00012	// LEFT DOOR OPEN
AND NOT   M06512	// L_2nd DIE VACUUM CHECK ON
OUT       M10614	// L_2nd DIE VC ALARM KP
; L176
LOADP     M00201	// LEFT AUTO RUN
OR        M1061A	// L_2nd DIE VC CLEAR OFF
AND       P00116	// L_2nd DIE VACUUM EJECTOR ON
OUT       M1061A	// L_2nd DIE VC CLEAR OFF
// ========== VACUUM ON/OFF ==========
; L179
LOAD NOT  M10580	// L_2nd MAND CYCLE RUN
AND NOT   M12080	// L_P&P CYCLE RUN
NOT
AND       M04022	// L_P&P Y PUT POS
AND       P00056	// L_P&P DOWN
AND       P00132	// L_P&P 2nd EJECT ON
ORP       T0050	// LF_AUTO RUN 0.05
AND NOT   P00116	// L_2nd DIE VACUUM EJECTOR ON
OR        M10822	// T)L_2nd VC ON
OR        M10620	// L_2nd MAND VC ON
AND NOT   M10622	// L_2nd MAND VC OFF
AND NOT   M10824	// T)L_2nd VC OFF
AND NOT   M1069F	// L_2nd MAND AUAc ¨ú©ª¨úiAu
AND NOT   M19102	// T)LEFT INITIAL
OUT       M10620	// L_2nd MAND VC ON

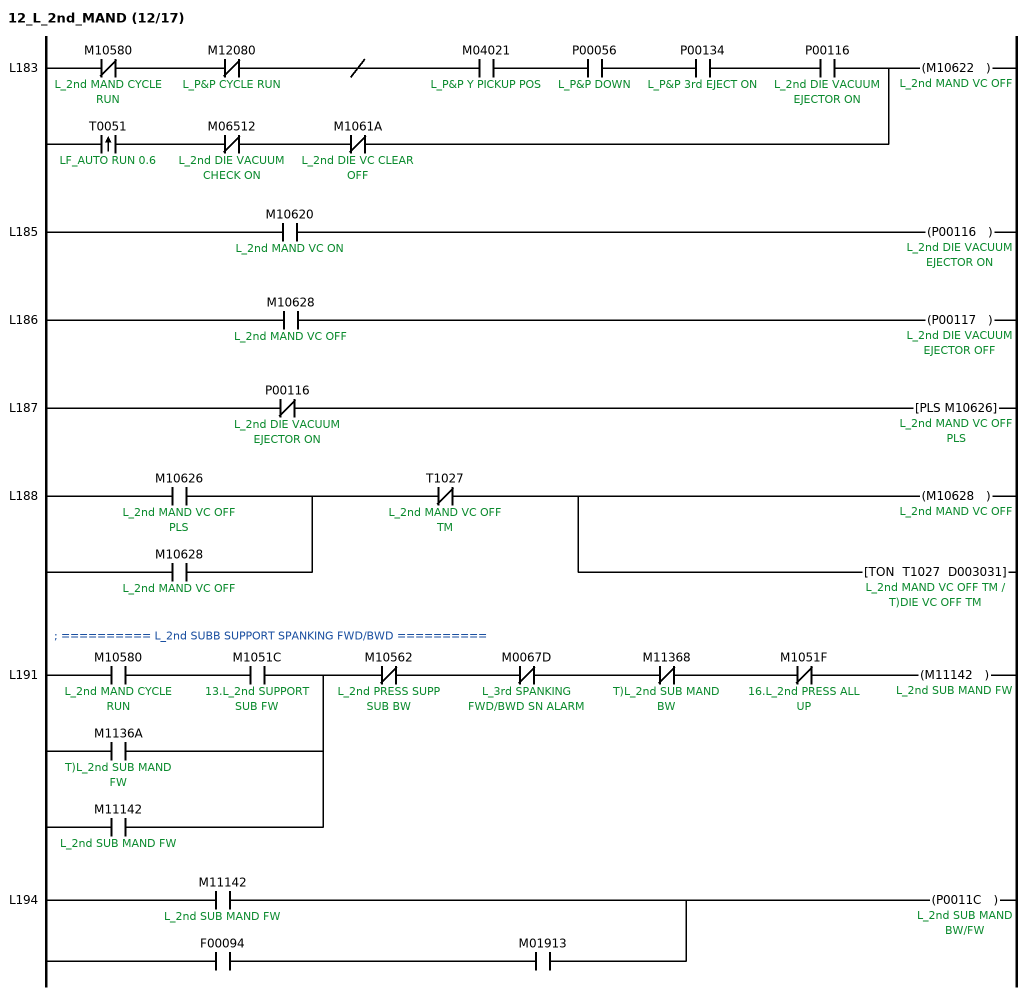
; L183
LOAD NOT  M10580	// L_2nd MAND CYCLE RUN
AND NOT   M12080	// L_P&P CYCLE RUN
NOT
AND       M04021	// L_P&P Y PICKUP POS
AND       P00056	// L_P&P DOWN
AND       P00134	// L_P&P 3rd EJECT ON
AND       P00116	// L_2nd DIE VACUUM EJECTOR ON
LOADP     T0051	// LF_AUTO RUN 0.6
AND NOT   M06512	// L_2nd DIE VACUUM CHECK ON
AND NOT   M1061A	// L_2nd DIE VC CLEAR OFF
OR LOAD
OUT       M10622	// L_2nd MAND VC OFF
; L185
LOAD      M10620	// L_2nd MAND VC ON
OUT       P00116	// L_2nd DIE VACUUM EJECTOR ON
; L186
LOAD      M10628	// L_2nd MAND VC OFF
OUT       P00117	// L_2nd DIE VACUUM EJECTOR OFF
; L187
LOAD NOT  P00116	// L_2nd DIE VACUUM EJECTOR ON
OUTP      M10626	// L_2nd MAND VC OFF PLS
; L188
LOAD      M10626	// L_2nd MAND VC OFF PLS
OR        M10628	// L_2nd MAND VC OFF
AND NOT   T1027	// L_2nd MAND VC OFF TM
OUT       M10628	// L_2nd MAND VC OFF
TON       T1027 D003031	// L_2nd MAND VC OFF TM / T)DIE VC OFF TM
// ========== L_2nd SUBB SUPPORT SPANKING FWD/BWD ==========
; L191
LOAD      M10580	// L_2nd MAND CYCLE RUN
AND       M1051C	// 13.L_2nd SUPPORT SUB FW
OR        M1136A	// T)L_2nd SUB MAND FW
OR        M11142	// L_2nd SUB MAND FW
AND NOT   M10562	// L_2nd PRESS SUPP SUB BW
AND NOT   M0067D	// L_3rd SPANKING FWD/BWD SN ALARM
AND NOT   M11368	// T)L_2nd SUB MAND BW
AND NOT   M1051F	// 16.L_2nd PRESS ALL UP
OUT       M11142	// L_2nd SUB MAND FW
; L194
LOAD      M11142	// L_2nd SUB MAND FW
LOAD      F00094
AND       M01913
OR LOAD
OUT       P0011C	// L_2nd SUB MAND BW/FW

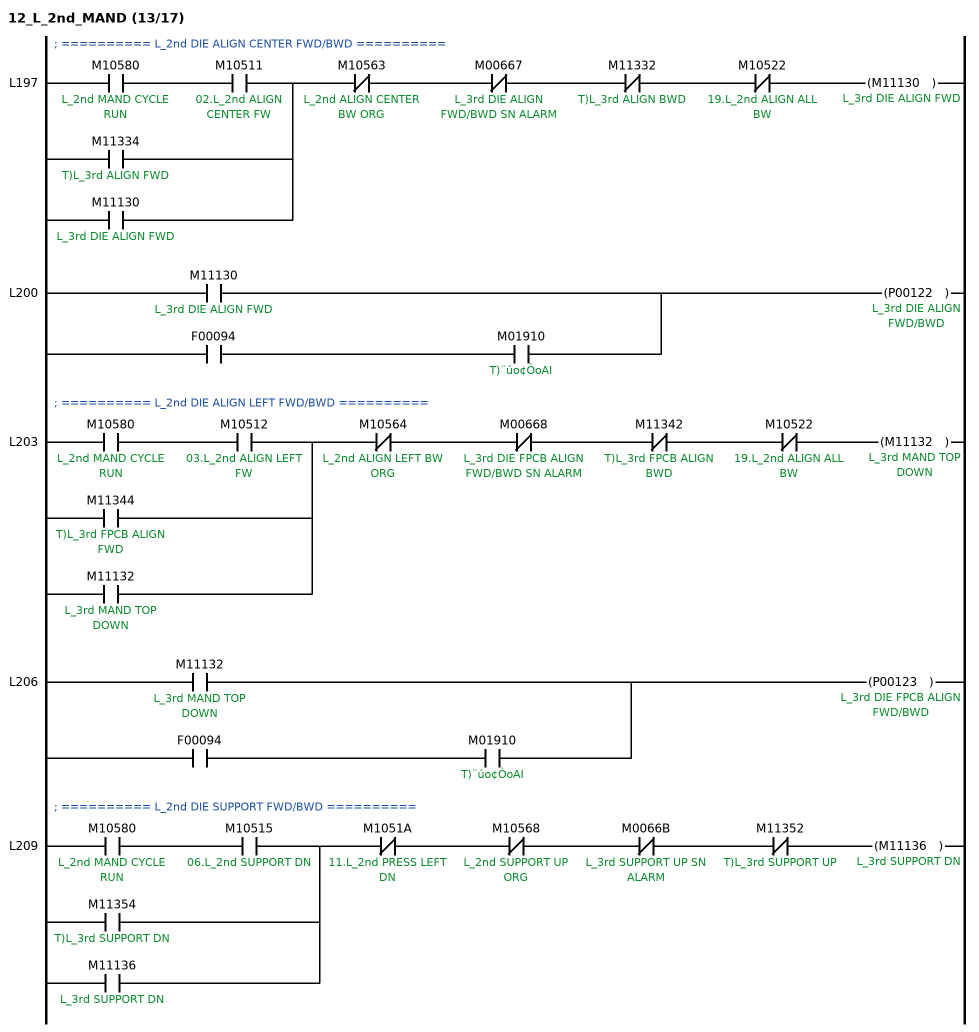
// ========== L_2nd DIE ALIGN CENTER FWD/BWD ==========
; L197
LOAD      M10580	// L_2nd MAND CYCLE RUN
AND       M10511	// 02.L_2nd ALIGN CENTER FW
OR        M11334	// T)L_3rd ALIGN FWD
OR        M11130	// L_3rd DIE ALIGN FWD
AND NOT   M10563	// L_2nd ALIGN CENTER BW ORG
AND NOT   M00667	// L_3rd DIE ALIGN FWD/BWD SN ALARM
AND NOT   M11332	// T)L_3rd ALIGN BWD
AND NOT   M10522	// 19.L_2nd ALIGN ALL BW
OUT       M11130	// L_3rd DIE ALIGN FWD
; L200
LOAD      M11130	// L_3rd DIE ALIGN FWD
LOAD      F00094
AND       M01910	// T)¨úo¢ÒoAI
OR LOAD
OUT       P00122	// L_3rd DIE ALIGN FWD/BWD
// ========== L_2nd DIE ALIGN LEFT FWD/BWD ==========
; L203
LOAD      M10580	// L_2nd MAND CYCLE RUN
AND       M10512	// 03.L_2nd ALIGN LEFT FW
OR        M11344	// T)L_3rd FPCB ALIGN FWD
OR        M11132	// L_3rd MAND TOP DOWN
AND NOT   M10564	// L_2nd ALIGN LEFT BW ORG
AND NOT   M00668	// L_3rd DIE FPCB ALIGN FWD/BWD SN ALARM
AND NOT   M11342	// T)L_3rd FPCB ALIGN BWD
AND NOT   M10522	// 19.L_2nd ALIGN ALL BW
OUT       M11132	// L_3rd MAND TOP DOWN
; L206
LOAD      M11132	// L_3rd MAND TOP DOWN
LOAD      F00094
AND       M01910	// T)¨úo¢ÒoAI
OR LOAD
OUT       P00123	// L_3rd DIE FPCB ALIGN FWD/BWD
// ========== L_2nd DIE SUPPORT FWD/BWD ==========
; L209
LOAD      M10580	// L_2nd MAND CYCLE RUN
AND       M10515	// 06.L_2nd SUPPORT DN
OR        M11354	// T)L_3rd SUPPORT DN
OR        M11136	// L_3rd SUPPORT DN
AND NOT   M1051A	// 11.L_2nd PRESS LEFT DN
AND NOT   M10568	// L_2nd SUPPORT UP ORG
AND NOT   M0066B	// L_3rd SUPPORT UP SN ALARM
AND NOT   M11352	// T)L_3rd SUPPORT UP
OUT       M11136	// L_3rd SUPPORT DN

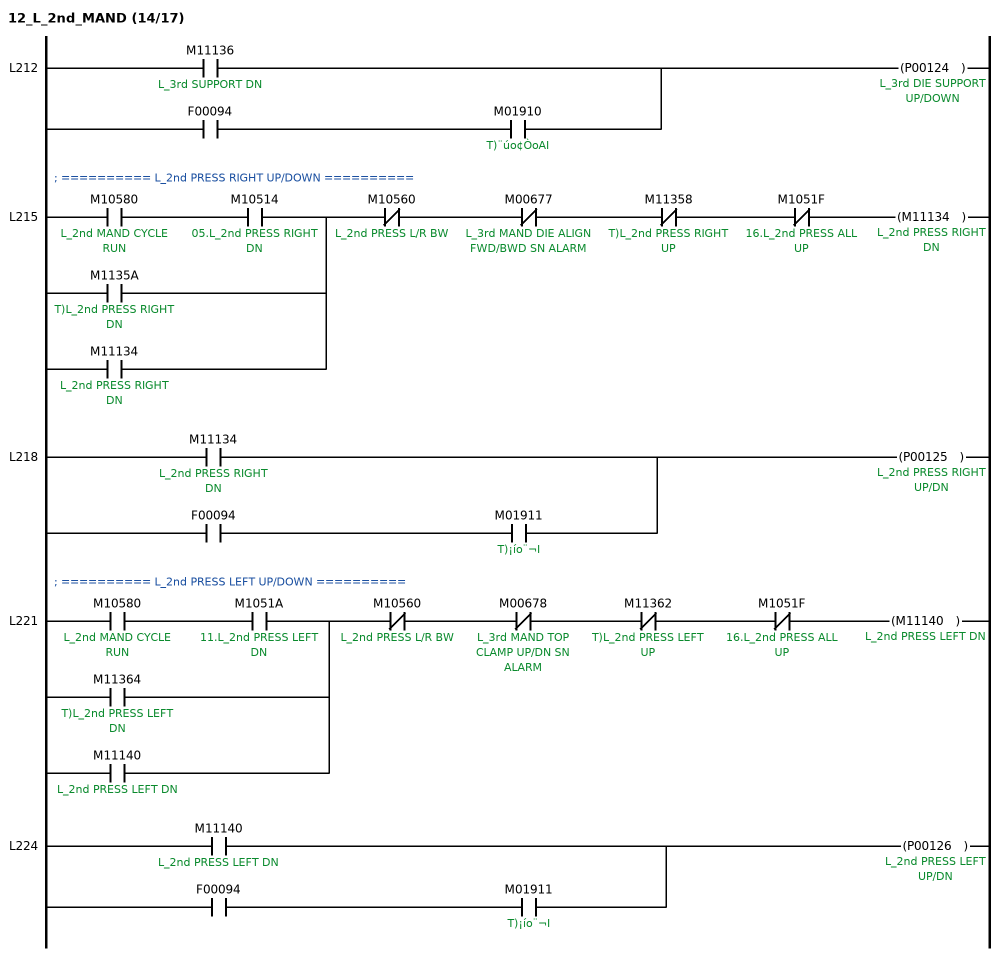
; L212
LOAD      M11136	// L_3rd SUPPORT DN
LOAD      F00094
AND       M01910	// T)¨úo¢ÒoAI
OR LOAD
OUT       P00124	// L_3rd DIE SUPPORT UP/DOWN
// ========== L_2nd PRESS RIGHT UP/DOWN ==========
; L215
LOAD      M10580	// L_2nd MAND CYCLE RUN
AND       M10514	// 05.L_2nd PRESS RIGHT DN
OR        M1135A	// T)L_2nd PRESS RIGHT DN
OR        M11134	// L_2nd PRESS RIGHT DN
AND NOT   M10560	// L_2nd PRESS L/R BW
AND NOT   M00677	// L_3rd MAND DIE ALIGN FWD/BWD SN ALARM
AND NOT   M11358	// T)L_2nd PRESS RIGHT UP
AND NOT   M1051F	// 16.L_2nd PRESS ALL UP
OUT       M11134	// L_2nd PRESS RIGHT DN
; L218
LOAD      M11134	// L_2nd PRESS RIGHT DN
LOAD      F00094
AND       M01911	// T)¡ío¨¬I
OR LOAD
OUT       P00125	// L_2nd PRESS RIGHT UP/DN
// ========== L_2nd PRESS LEFT UP/DOWN ==========
; L221
LOAD      M10580	// L_2nd MAND CYCLE RUN
AND       M1051A	// 11.L_2nd PRESS LEFT DN
OR        M11364	// T)L_2nd PRESS LEFT DN
OR        M11140	// L_2nd PRESS LEFT DN
AND NOT   M10560	// L_2nd PRESS L/R BW
AND NOT   M00678	// L_3rd MAND TOP CLAMP UP/DN SN ALARM
AND NOT   M11362	// T)L_2nd PRESS LEFT UP
AND NOT   M1051F	// 16.L_2nd PRESS ALL UP
OUT       M11140	// L_2nd PRESS LEFT DN
; L224
LOAD      M11140	// L_2nd PRESS LEFT DN
LOAD      F00094
AND       M01911	// T)¡ío¨¬I
OR LOAD
OUT       P00126	// L_2nd PRESS LEFT UP/DN

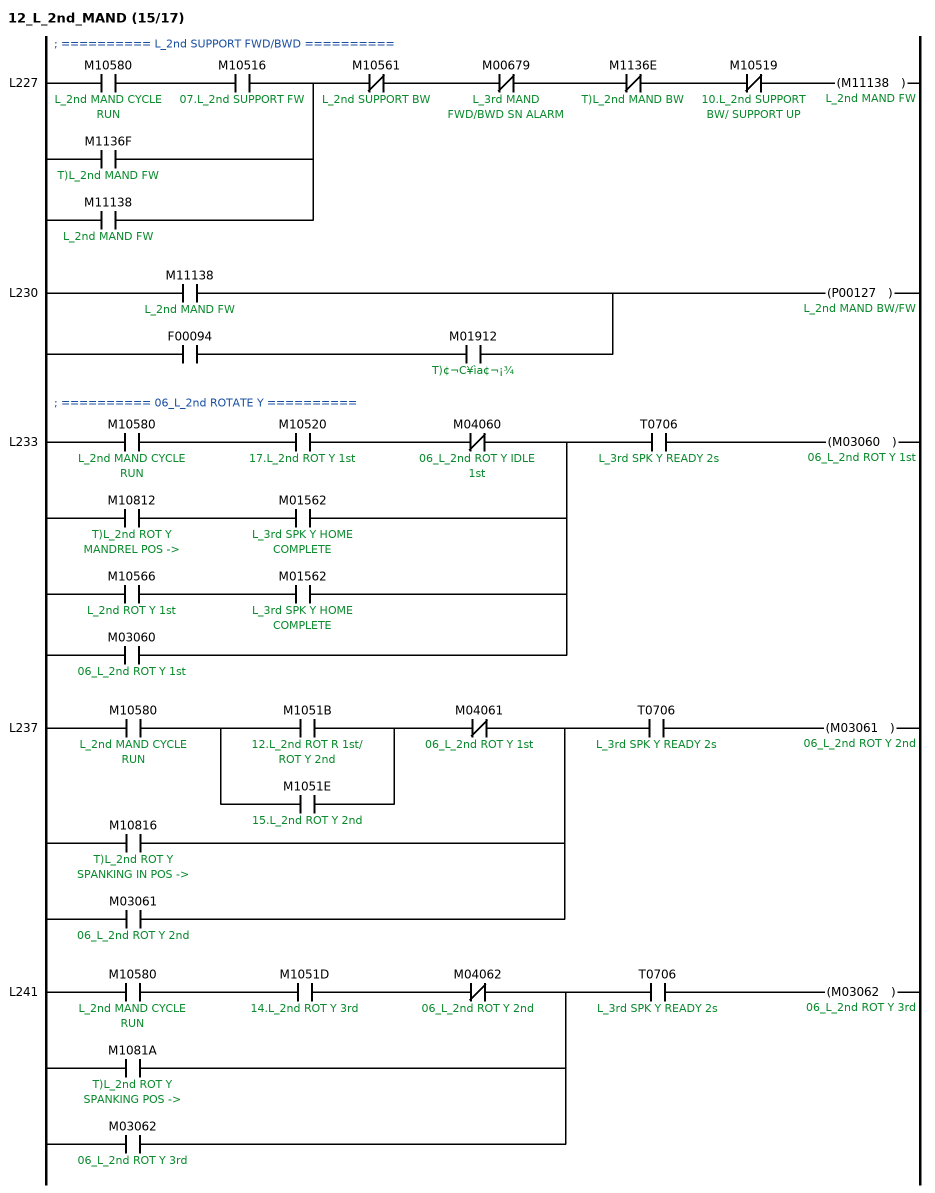
// ========== L_2nd SUPPORT FWD/BWD ==========
; L227
LOAD      M10580	// L_2nd MAND CYCLE RUN
AND       M10516	// 07.L_2nd SUPPORT FW
OR        M1136F	// T)L_2nd MAND FW
OR        M11138	// L_2nd MAND FW
AND NOT   M10561	// L_2nd SUPPORT BW
AND NOT   M00679	// L_3rd MAND FWD/BWD SN ALARM
AND NOT   M1136E	// T)L_2nd MAND BW
AND NOT   M10519	// 10.L_2nd SUPPORT BW/ SUPPORT UP
OUT       M11138	// L_2nd MAND FW
; L230
LOAD      M11138	// L_2nd MAND FW
LOAD      F00094
AND       M01912	// T)¢¬C¥ìa¢¬¡¾
OR LOAD
OUT       P00127	// L_2nd MAND BW/FW
// ========== 06_L_2nd ROTATE Y ==========
; L233
LOAD      M10580	// L_2nd MAND CYCLE RUN
AND       M10520	// 17.L_2nd ROT Y 1st
AND NOT   M04060	// 06_L_2nd ROT Y IDLE 1st
LOAD      M10812	// T)L_2nd ROT Y MANDREL POS ->
AND       M01562	// L_3rd SPK Y HOME COMPLETE
OR LOAD
LOAD      M10566	// L_2nd ROT Y 1st
AND       M01562	// L_3rd SPK Y HOME COMPLETE
OR LOAD
OR        M03060	// 06_L_2nd ROT Y 1st
AND       T0706	// L_3rd SPK Y READY 2s
OUT       M03060	// 06_L_2nd ROT Y 1st
; L237
LOAD      M10580	// L_2nd MAND CYCLE RUN
LOAD      M1051B	// 12.L_2nd ROT R 1st/ ROT Y 2nd
OR        M1051E	// 15.L_2nd ROT Y 2nd
AND LOAD
AND NOT   M04061	// 06_L_2nd ROT Y 1st
OR        M10816	// T)L_2nd ROT Y SPANKING IN POS ->
OR        M03061	// 06_L_2nd ROT Y 2nd
AND       T0706	// L_3rd SPK Y READY 2s
OUT       M03061	// 06_L_2nd ROT Y 2nd
; L241
LOAD      M10580	// L_2nd MAND CYCLE RUN
AND       M1051D	// 14.L_2nd ROT Y 3rd
AND NOT   M04062	// 06_L_2nd ROT Y 2nd
OR        M1081A	// T)L_2nd ROT Y SPANKING POS ->
OR        M03062	// 06_L_2nd ROT Y 3rd
AND       T0706	// L_3rd SPK Y READY 2s
OUT       M03062	// 06_L_2nd ROT Y 3rd

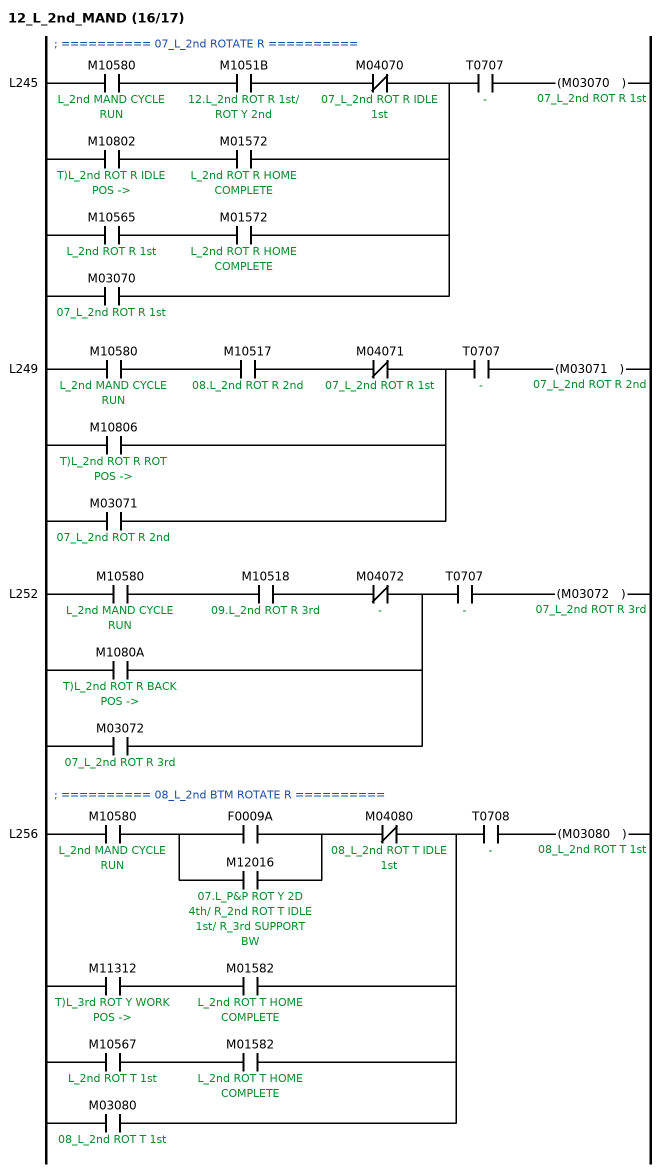
// ========== 07_L_2nd ROTATE R ==========
; L245
LOAD      M10580	// L_2nd MAND CYCLE RUN
AND       M1051B	// 12.L_2nd ROT R 1st/ ROT Y 2nd
AND NOT   M04070	// 07_L_2nd ROT R IDLE 1st
LOAD      M10802	// T)L_2nd ROT R IDLE POS ->
AND       M01572	// L_2nd ROT R HOME COMPLETE
OR LOAD
LOAD      M10565	// L_2nd ROT R 1st
AND       M01572	// L_2nd ROT R HOME COMPLETE
OR LOAD
OR        M03070	// 07_L_2nd ROT R 1st
AND       T0707	// -
OUT       M03070	// 07_L_2nd ROT R 1st
; L249
LOAD      M10580	// L_2nd MAND CYCLE RUN
AND       M10517	// 08.L_2nd ROT R 2nd
AND NOT   M04071	// 07_L_2nd ROT R 1st
OR        M10806	// T)L_2nd ROT R ROT POS ->
OR        M03071	// 07_L_2nd ROT R 2nd
AND       T0707	// -
OUT       M03071	// 07_L_2nd ROT R 2nd
; L252
LOAD      M10580	// L_2nd MAND CYCLE RUN
AND       M10518	// 09.L_2nd ROT R 3rd
AND NOT   M04072	// -
OR        M1080A	// T)L_2nd ROT R BACK POS ->
OR        M03072	// 07_L_2nd ROT R 3rd
AND       T0707	// -
OUT       M03072	// 07_L_2nd ROT R 3rd
// ========== 08_L_2nd BTM ROTATE R ==========
; L256
LOAD      M10580	// L_2nd MAND CYCLE RUN
LOAD      F0009A
OR        M12016	// 07.L_P&P ROT Y 2D 4th/ R_2nd ROT T IDLE 1st/ R_3rd SUPPORT BW
AND LOAD
AND NOT   M04080	// 08_L_2nd ROT T IDLE 1st
LOAD      M11312	// T)L_3rd ROT Y WORK POS ->
AND       M01582	// L_2nd ROT T HOME COMPLETE
OR LOAD
LOAD      M10567	// L_2nd ROT T 1st
AND       M01582	// L_2nd ROT T HOME COMPLETE
OR LOAD
OR        M03080	// 08_L_2nd ROT T 1st
AND       T0708	// -
OUT       M03080	// 08_L_2nd ROT T 1st

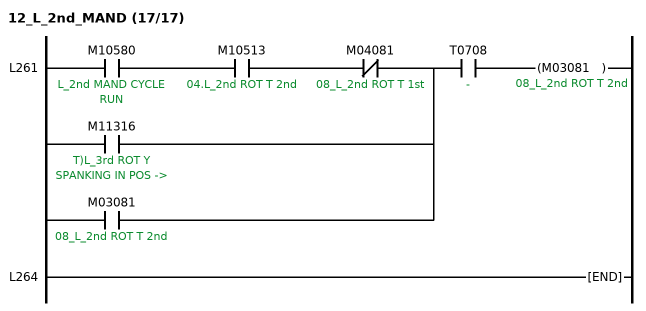
; L261
LOAD      M10580	// L_2nd MAND CYCLE RUN
AND       M10513	// 04.L_2nd ROT T 2nd
AND NOT   M04081	// 08_L_2nd ROT T 1st
OR        M11316	// T)L_3rd ROT Y SPANKING IN POS ->
OR        M03081	// 08_L_2nd ROT T 2nd
AND       T0708	// -
OUT       M03081	// 08_L_2nd ROT T 2nd
; L264
END

PROGRAM 13_L_3rd_MAND (task: ¨ö¨¬A¥ì CA¡¤I¡¾¡¿¡¤¡Í)

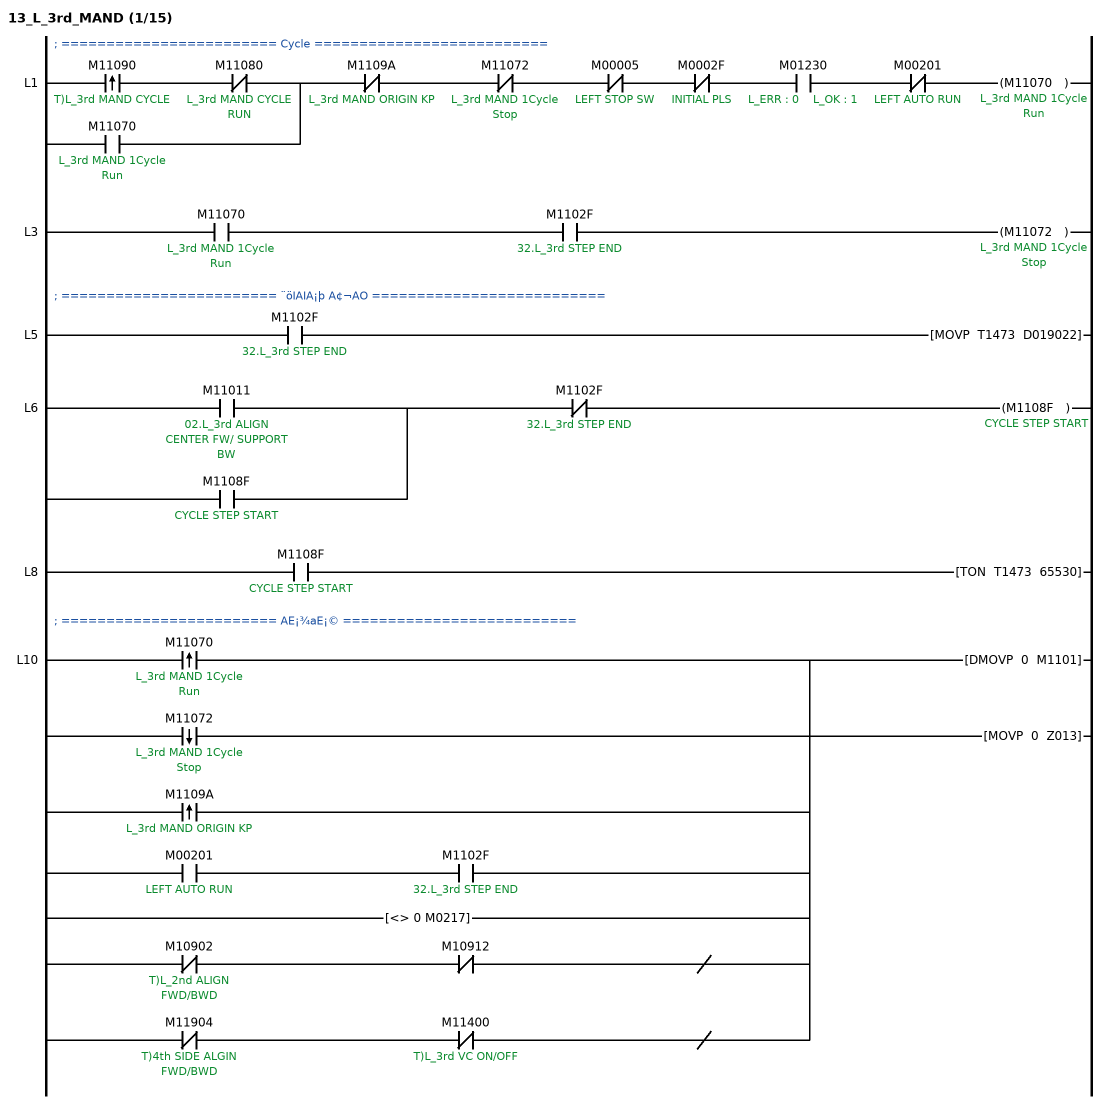
// ======================== Cycle ==========================
; L1
LOADP     M11090	// T)L_3rd MAND CYCLE
AND NOT   M11080	// L_3rd MAND CYCLE RUN
OR        M11070	// L_3rd MAND 1Cycle Run
AND NOT   M1109A	// L_3rd MAND ORIGIN KP
AND NOT   M11072	// L_3rd MAND 1Cycle Stop
AND NOT   M00005	// LEFT STOP SW
AND NOT   M0002F	// INITIAL PLS
AND       M01230	// L_ERR : 0    L_OK : 1
AND NOT   M00201	// LEFT AUTO RUN
OUT       M11070	// L_3rd MAND 1Cycle Run
; L3
LOAD      M11070	// L_3rd MAND 1Cycle Run
AND       M1102F	// 32.L_3rd STEP END
OUT       M11072	// L_3rd MAND 1Cycle Stop
// ======================== ¨öIAIA¡þ A¢¬AO ==========================
; L5
LOAD      M1102F	// 32.L_3rd STEP END
MOVP      T1473 D019022
; L6
LOAD      M11011	// 02.L_3rd ALIGN CENTER FW/ SUPPORT BW
OR        M1108F	// CYCLE STEP START
AND NOT   M1102F	// 32.L_3rd STEP END
OUT       M1108F	// CYCLE STEP START
; L8
LOAD      M1108F	// CYCLE STEP START
TON       T1473 65530
// ======================== AE¡¾aE¡© ==========================
; L10
LOADP     M11070	// L_3rd MAND 1Cycle Run
ORN       M11072	// L_3rd MAND 1Cycle Stop
ORP       M1109A	// L_3rd MAND ORIGIN KP
LOAD      M00201	// LEFT AUTO RUN
AND       M1102F	// 32.L_3rd STEP END
OR LOAD
OR<>      0 M0217
LOAD NOT  M10902	// T)L_2nd ALIGN FWD/BWD
AND NOT   M10912
NOT
OR LOAD
LOAD NOT  M11904	// T)4th SIDE ALGIN FWD/BWD
AND NOT   M11400	// T)L_3rd VC ON/OFF
NOT
OR LOAD
DMOVP     0 M1101
MOVP      0 Z013

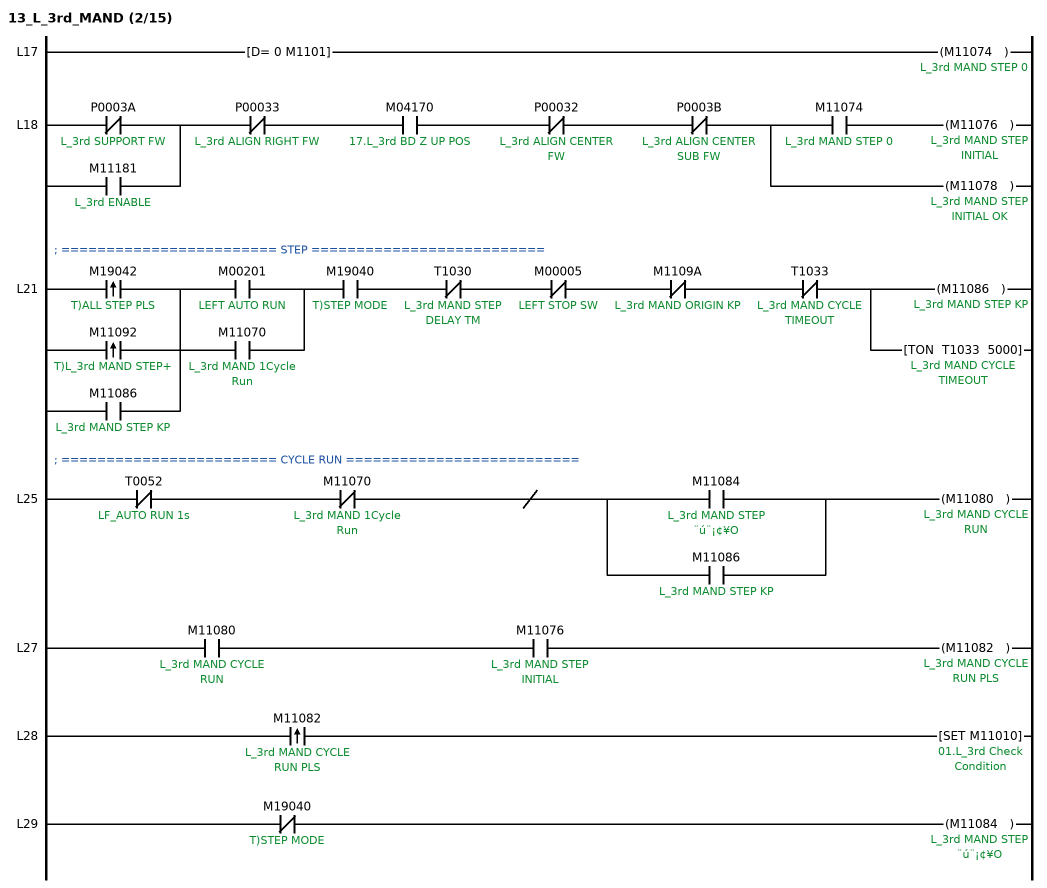
; L17
LOADD=    0 M1101
OUT       M11074	// L_3rd MAND STEP 0
; L18
LOAD NOT  P0003A	// L_3rd SUPPORT FW
OR        M11181	// L_3rd ENABLE
AND NOT   P00033	// L_3rd ALIGN RIGHT FW
AND       M04170	// 17.L_3rd BD Z UP POS
AND NOT   P00032	// L_3rd ALIGN CENTER FW
AND NOT   P0003B	// L_3rd ALIGN CENTER SUB FW
MPUSH
AND       M11074	// L_3rd MAND STEP 0
OUT       M11076	// L_3rd MAND STEP INITIAL
MPOP
OUT       M11078	// L_3rd MAND STEP INITIAL OK
// ======================== STEP ==========================
; L21
LOADP     M19042	// T)ALL STEP PLS
ORP       M11092	// T)L_3rd MAND STEP+
OR        M11086	// L_3rd MAND STEP KP
LOAD      M00201	// LEFT AUTO RUN
OR        M11070	// L_3rd MAND 1Cycle Run
AND LOAD
AND       M19040	// T)STEP MODE
AND NOT   T1030	// L_3rd MAND STEP DELAY TM
AND NOT   M00005	// LEFT STOP SW
AND NOT   M1109A	// L_3rd MAND ORIGIN KP
AND NOT   T1033	// L_3rd MAND CYCLE TIMEOUT
OUT       M11086	// L_3rd MAND STEP KP
TON       T1033 5000	// L_3rd MAND CYCLE TIMEOUT
// ======================== CYCLE RUN ==========================
; L25
LOAD NOT  T0052	// LF_AUTO RUN 1s
AND NOT   M11070	// L_3rd MAND 1Cycle Run
NOT
LOAD      M11084	// L_3rd MAND STEP ¨ú¨¡¢¥O
OR        M11086	// L_3rd MAND STEP KP
AND LOAD
OUT       M11080	// L_3rd MAND CYCLE RUN
; L27
LOAD      M11080	// L_3rd MAND CYCLE RUN
AND       M11076	// L_3rd MAND STEP INITIAL
OUT       M11082	// L_3rd MAND CYCLE RUN PLS
; L28
LOADP     M11082	// L_3rd MAND CYCLE RUN PLS
SET       M11010	// 01.L_3rd Check Condition
; L29
LOAD NOT  M19040	// T)STEP MODE
OUT       M11084	// L_3rd MAND STEP ¨ú¨¡¢¥O

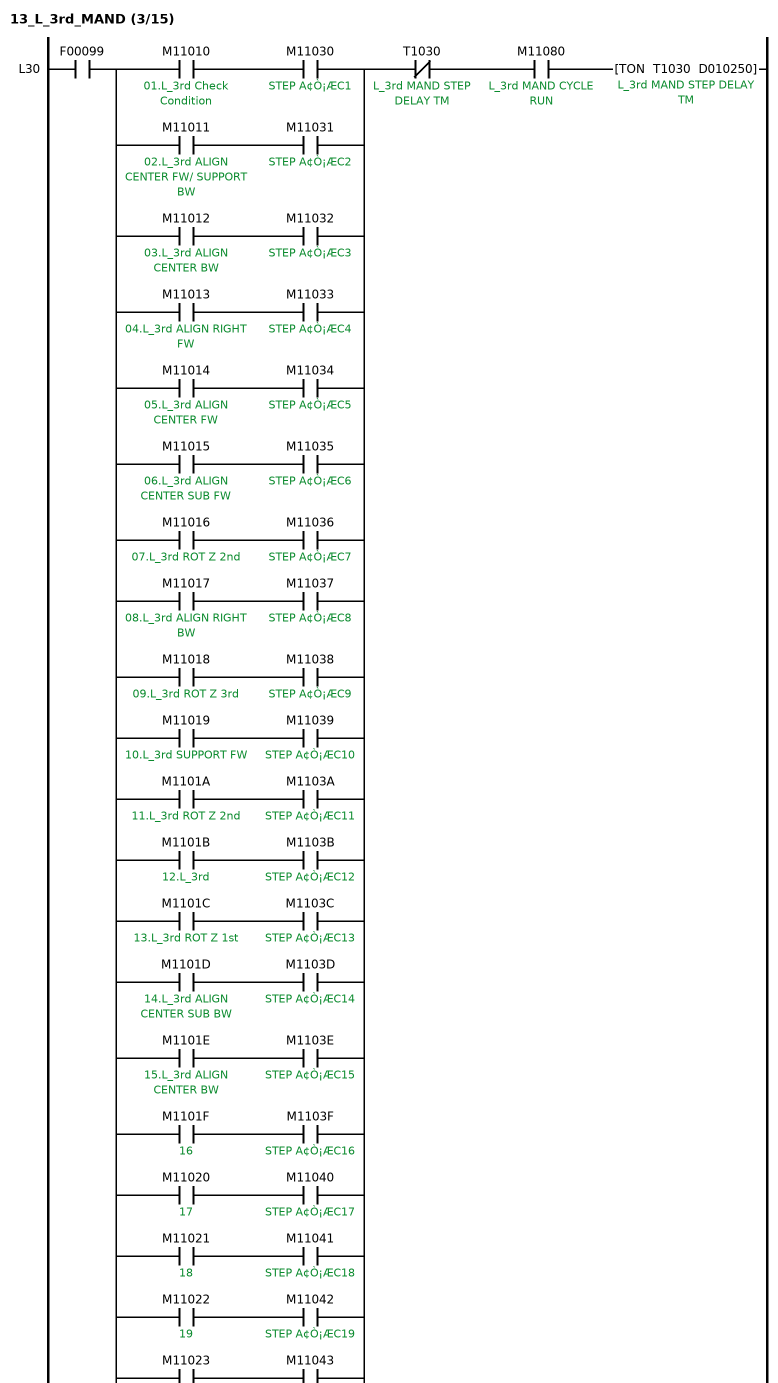

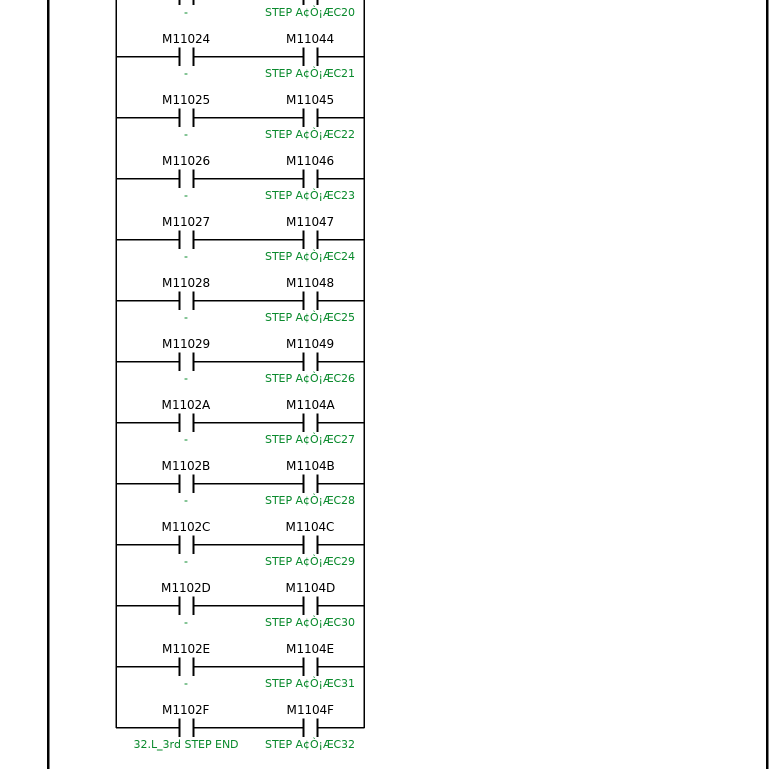
; L30
LOAD      F00099
LOAD      M11010	// 01.L_3rd Check Condition
AND       M11030	// STEP A¢Ò¡ÆC1
LOAD      M11011	// 02.L_3rd ALIGN CENTER FW/ SUPPORT BW
AND       M11031	// STEP A¢Ò¡ÆC2
OR LOAD
LOAD      M11012	// 03.L_3rd ALIGN CENTER BW
AND       M11032	// STEP A¢Ò¡ÆC3
OR LOAD
LOAD      M11013	// 04.L_3rd ALIGN RIGHT FW
AND       M11033	// STEP A¢Ò¡ÆC4
OR LOAD
LOAD      M11014	// 05.L_3rd ALIGN CENTER FW
AND       M11034	// STEP A¢Ò¡ÆC5
OR LOAD
LOAD      M11015	// 06.L_3rd ALIGN CENTER SUB FW
AND       M11035	// STEP A¢Ò¡ÆC6
OR LOAD
LOAD      M11016	// 07.L_3rd ROT Z 2nd
AND       M11036	// STEP A¢Ò¡ÆC7
OR LOAD
LOAD      M11017	// 08.L_3rd ALIGN RIGHT BW
AND       M11037	// STEP A¢Ò¡ÆC8
OR LOAD
LOAD      M11018	// 09.L_3rd ROT Z 3rd
AND       M11038	// STEP A¢Ò¡ÆC9
OR LOAD
LOAD      M11019	// 10.L_3rd SUPPORT FW
AND       M11039	// STEP A¢Ò¡ÆC10
OR LOAD
LOAD      M1101A	// 11.L_3rd ROT Z 2nd
AND       M1103A	// STEP A¢Ò¡ÆC11
OR LOAD
LOAD      M1101B	// 12.L_3rd 
AND       M1103B	// STEP A¢Ò¡ÆC12
OR LOAD
LOAD      M1101C	// 13.L_3rd ROT Z 1st
AND       M1103C	// STEP A¢Ò¡ÆC13
OR LOAD
LOAD      M1101D	// 14.L_3rd ALIGN CENTER SUB BW
AND       M1103D	// STEP A¢Ò¡ÆC14
OR LOAD
LOAD      M1101E	// 15.L_3rd ALIGN CENTER BW
AND       M1103E	// STEP A¢Ò¡ÆC15
OR LOAD
LOAD      M1101F	// 16
AND       M1103F	// STEP A¢Ò¡ÆC16
OR LOAD
LOAD      M11020	// 17
AND       M11040	// STEP A¢Ò¡ÆC17
OR LOAD
LOAD      M11021	// 18
AND       M11041	// STEP A¢Ò¡ÆC18
OR LOAD
LOAD      M11022	// 19
AND       M11042	// STEP A¢Ò¡ÆC19
OR LOAD
LOAD      M11023	// -
AND       M11043	// STEP A¢Ò¡ÆC20
OR LOAD
LOAD      M11024	// -
AND       M11044	// STEP A¢Ò¡ÆC21
OR LOAD
LOAD      M11025	// -
AND       M11045	// STEP A¢Ò¡ÆC22
OR LOAD
LOAD      M11026	// -
AND       M11046	// STEP A¢Ò¡ÆC23
OR LOAD
LOAD      M11027	// -
AND       M11047	// STEP A¢Ò¡ÆC24
OR LOAD
LOAD      M11028	// -
AND       M11048	// STEP A¢Ò¡ÆC25
OR LOAD
LOAD      M11029	// -
AND       M11049	// STEP A¢Ò¡ÆC26
OR LOAD
LOAD      M1102A	// -
AND       M1104A	// STEP A¢Ò¡ÆC27
OR LOAD
LOAD      M1102B	// -
AND       M1104B	// STEP A¢Ò¡ÆC28
OR LOAD
LOAD      M1102C	// -
AND       M1104C	// STEP A¢Ò¡ÆC29
OR LOAD
LOAD      M1102D	// -
AND       M1104D	// STEP A¢Ò¡ÆC30
OR LOAD
LOAD      M1102E	// -
AND       M1104E	// STEP A¢Ò¡ÆC31
OR LOAD
LOAD      M1102F	// 32.L_3rd STEP END
AND       M1104F	// STEP A¢Ò¡ÆC32
OR LOAD
AND LOAD
AND NOT   T1030	// L_3rd MAND STEP DELAY TM
AND       M11080	// L_3rd MAND CYCLE RUN
TON       T1030 D010250	// L_3rd MAND STEP DELAY TM

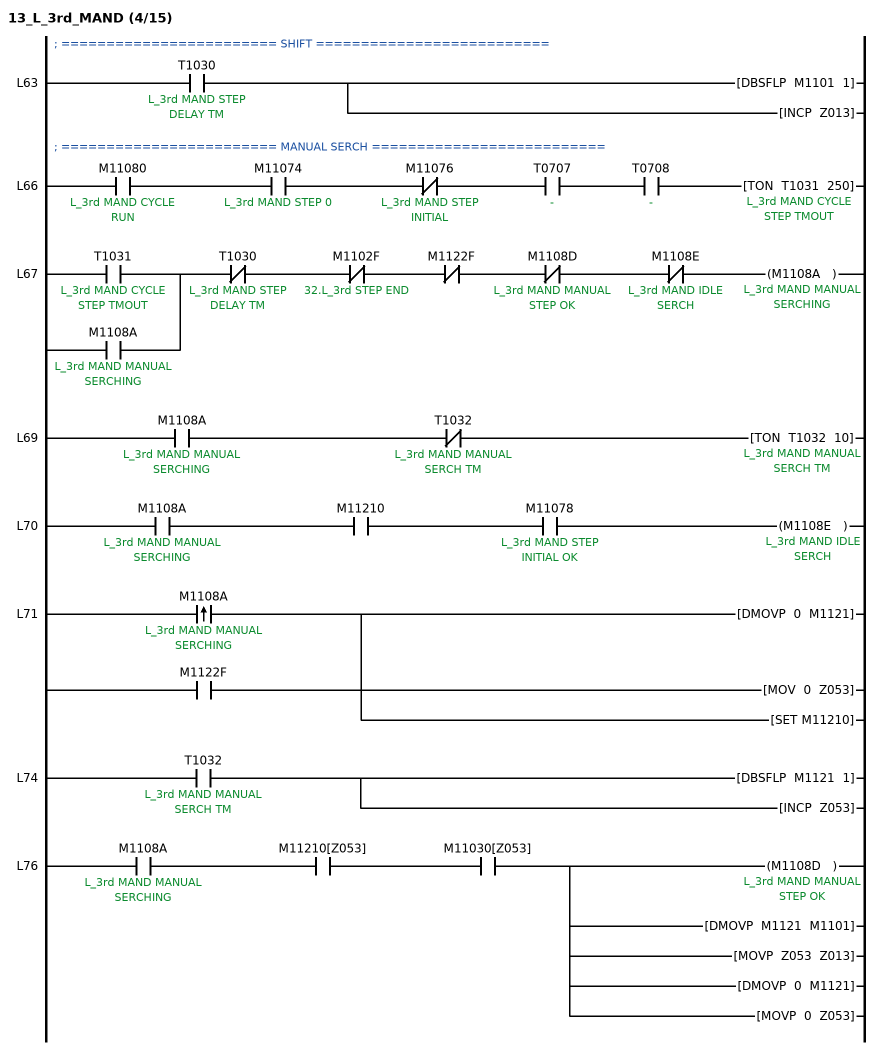
// ======================== SHIFT ==========================
; L63
LOAD      T1030	// L_3rd MAND STEP DELAY TM
DBSFLP    M1101 1
INCP      Z013
// ======================== MANUAL SERCH ==========================
; L66
LOAD      M11080	// L_3rd MAND CYCLE RUN
AND       M11074	// L_3rd MAND STEP 0
AND NOT   M11076	// L_3rd MAND STEP INITIAL
AND       T0707	// -
AND       T0708	// -
TON       T1031 250	// L_3rd MAND CYCLE STEP TMOUT
; L67
LOAD      T1031	// L_3rd MAND CYCLE STEP TMOUT
OR        M1108A	// L_3rd MAND MANUAL SERCHING
AND NOT   T1030	// L_3rd MAND STEP DELAY TM
AND NOT   M1102F	// 32.L_3rd STEP END
AND NOT   M1122F
AND NOT   M1108D	// L_3rd MAND MANUAL STEP OK
AND NOT   M1108E	// L_3rd MAND IDLE SERCH
OUT       M1108A	// L_3rd MAND MANUAL SERCHING
; L69
LOAD      M1108A	// L_3rd MAND MANUAL SERCHING
AND NOT   T1032	// L_3rd MAND MANUAL SERCH TM
TON       T1032 10	// L_3rd MAND MANUAL SERCH TM
; L70
LOAD      M1108A	// L_3rd MAND MANUAL SERCHING
AND       M11210
AND       M11078	// L_3rd MAND STEP INITIAL OK
OUT       M1108E	// L_3rd MAND IDLE SERCH
; L71
LOADP     M1108A	// L_3rd MAND MANUAL SERCHING
OR        M1122F
DMOVP     0 M1121
MOV       0 Z053
SET       M11210
; L74
LOAD      T1032	// L_3rd MAND MANUAL SERCH TM
DBSFLP    M1121 1
INCP      Z053
; L76
LOAD      M1108A	// L_3rd MAND MANUAL SERCHING
AND       M11210[Z053]
AND       M11030[Z053]
OUT       M1108D	// L_3rd MAND MANUAL STEP OK
DMOVP     M1121 M1101
MOVP      Z053 Z013
DMOVP     0 M1121
MOVP      0 Z053

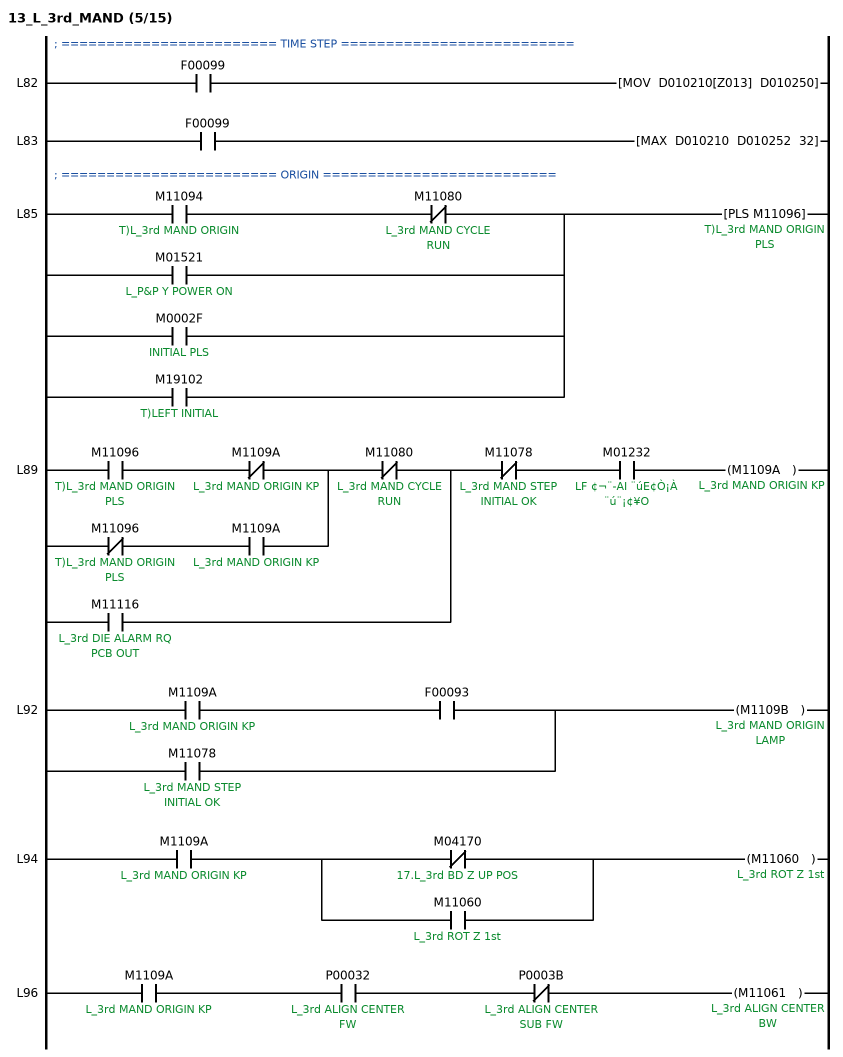
// ======================== TIME STEP ==========================
; L82
LOAD      F00099
MOV       D010210[Z013] D010250
; L83
LOAD      F00099
MAX       D010210 D010252 32
// ======================== ORIGIN ==========================
; L85
LOAD      M11094	// T)L_3rd MAND ORIGIN
AND NOT   M11080	// L_3rd MAND CYCLE RUN
OR        M01521	// L_P&P Y POWER ON
OR        M0002F	// INITIAL PLS
OR        M19102	// T)LEFT INITIAL
OUTP      M11096	// T)L_3rd MAND ORIGIN PLS
; L89
LOAD      M11096	// T)L_3rd MAND ORIGIN PLS
AND NOT   M1109A	// L_3rd MAND ORIGIN KP
LOAD NOT  M11096	// T)L_3rd MAND ORIGIN PLS
AND       M1109A	// L_3rd MAND ORIGIN KP
OR LOAD
AND NOT   M11080	// L_3rd MAND CYCLE RUN
OR        M11116	// L_3rd DIE ALARM RQ PCB OUT
AND NOT   M11078	// L_3rd MAND STEP INITIAL OK
AND       M01232	// LF ¢¬¨­AI ¨úE¢Ò¡À ¨ú¨¡¢¥O
OUT       M1109A	// L_3rd MAND ORIGIN KP
; L92
LOAD      M1109A	// L_3rd MAND ORIGIN KP
AND       F00093
OR        M11078	// L_3rd MAND STEP INITIAL OK
OUT       M1109B	// L_3rd MAND ORIGIN LAMP
; L94
LOAD      M1109A	// L_3rd MAND ORIGIN KP
LOAD NOT  M04170	// 17.L_3rd BD Z UP POS
OR        M11060	// L_3rd ROT Z 1st
AND LOAD
OUT       M11060	// L_3rd ROT Z 1st
; L96
LOAD      M1109A	// L_3rd MAND ORIGIN KP
AND       P00032	// L_3rd ALIGN CENTER FW
AND NOT   P0003B	// L_3rd ALIGN CENTER SUB FW
OUT       M11061	// L_3rd ALIGN CENTER BW

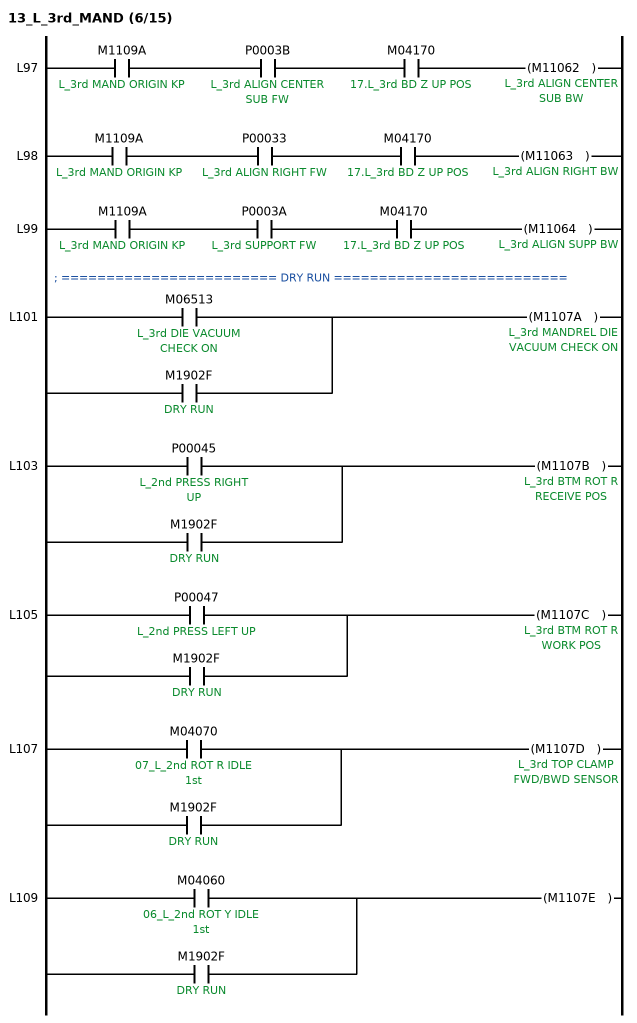
; L97
LOAD      M1109A	// L_3rd MAND ORIGIN KP
AND       P0003B	// L_3rd ALIGN CENTER SUB FW
AND       M04170	// 17.L_3rd BD Z UP POS
OUT       M11062	// L_3rd ALIGN CENTER SUB BW
; L98
LOAD      M1109A	// L_3rd MAND ORIGIN KP
AND       P00033	// L_3rd ALIGN RIGHT FW
AND       M04170	// 17.L_3rd BD Z UP POS
OUT       M11063	// L_3rd ALIGN RIGHT BW
; L99
LOAD      M1109A	// L_3rd MAND ORIGIN KP
AND       P0003A	// L_3rd SUPPORT FW
AND       M04170	// 17.L_3rd BD Z UP POS
OUT       M11064	// L_3rd ALIGN SUPP BW
// ======================== DRY RUN ==========================
; L101
LOAD      M06513	// L_3rd DIE VACUUM CHECK ON
OR        M1902F	// DRY RUN
OUT       M1107A	// L_3rd MANDREL DIE VACUUM CHECK ON
; L103
LOAD      P00045	// L_2nd PRESS RIGHT UP
OR        M1902F	// DRY RUN
OUT       M1107B	// L_3rd BTM ROT R RECEIVE POS
; L105
LOAD      P00047	// L_2nd PRESS LEFT UP
OR        M1902F	// DRY RUN
OUT       M1107C	// L_3rd BTM ROT R WORK POS
; L107
LOAD      M04070	// 07_L_2nd ROT R IDLE 1st
OR        M1902F	// DRY RUN
OUT       M1107D	// L_3rd TOP CLAMP FWD/BWD SENSOR
; L109
LOAD      M04060	// 06_L_2nd ROT Y IDLE 1st
OR        M1902F	// DRY RUN
OUT       M1107E

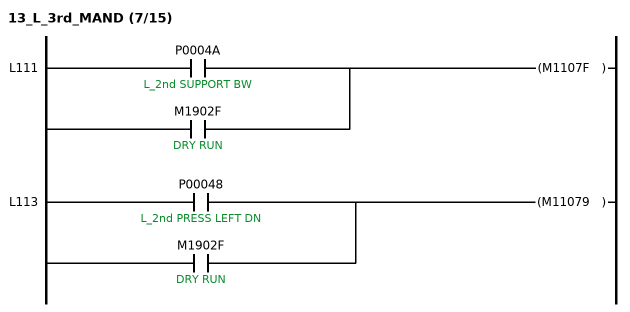
; L111
LOAD      P0004A	// L_2nd SUPPORT BW
OR        M1902F	// DRY RUN
OUT       M1107F
; L113
LOAD      P00048	// L_2nd PRESS LEFT DN
OR        M1902F	// DRY RUN
OUT       M11079

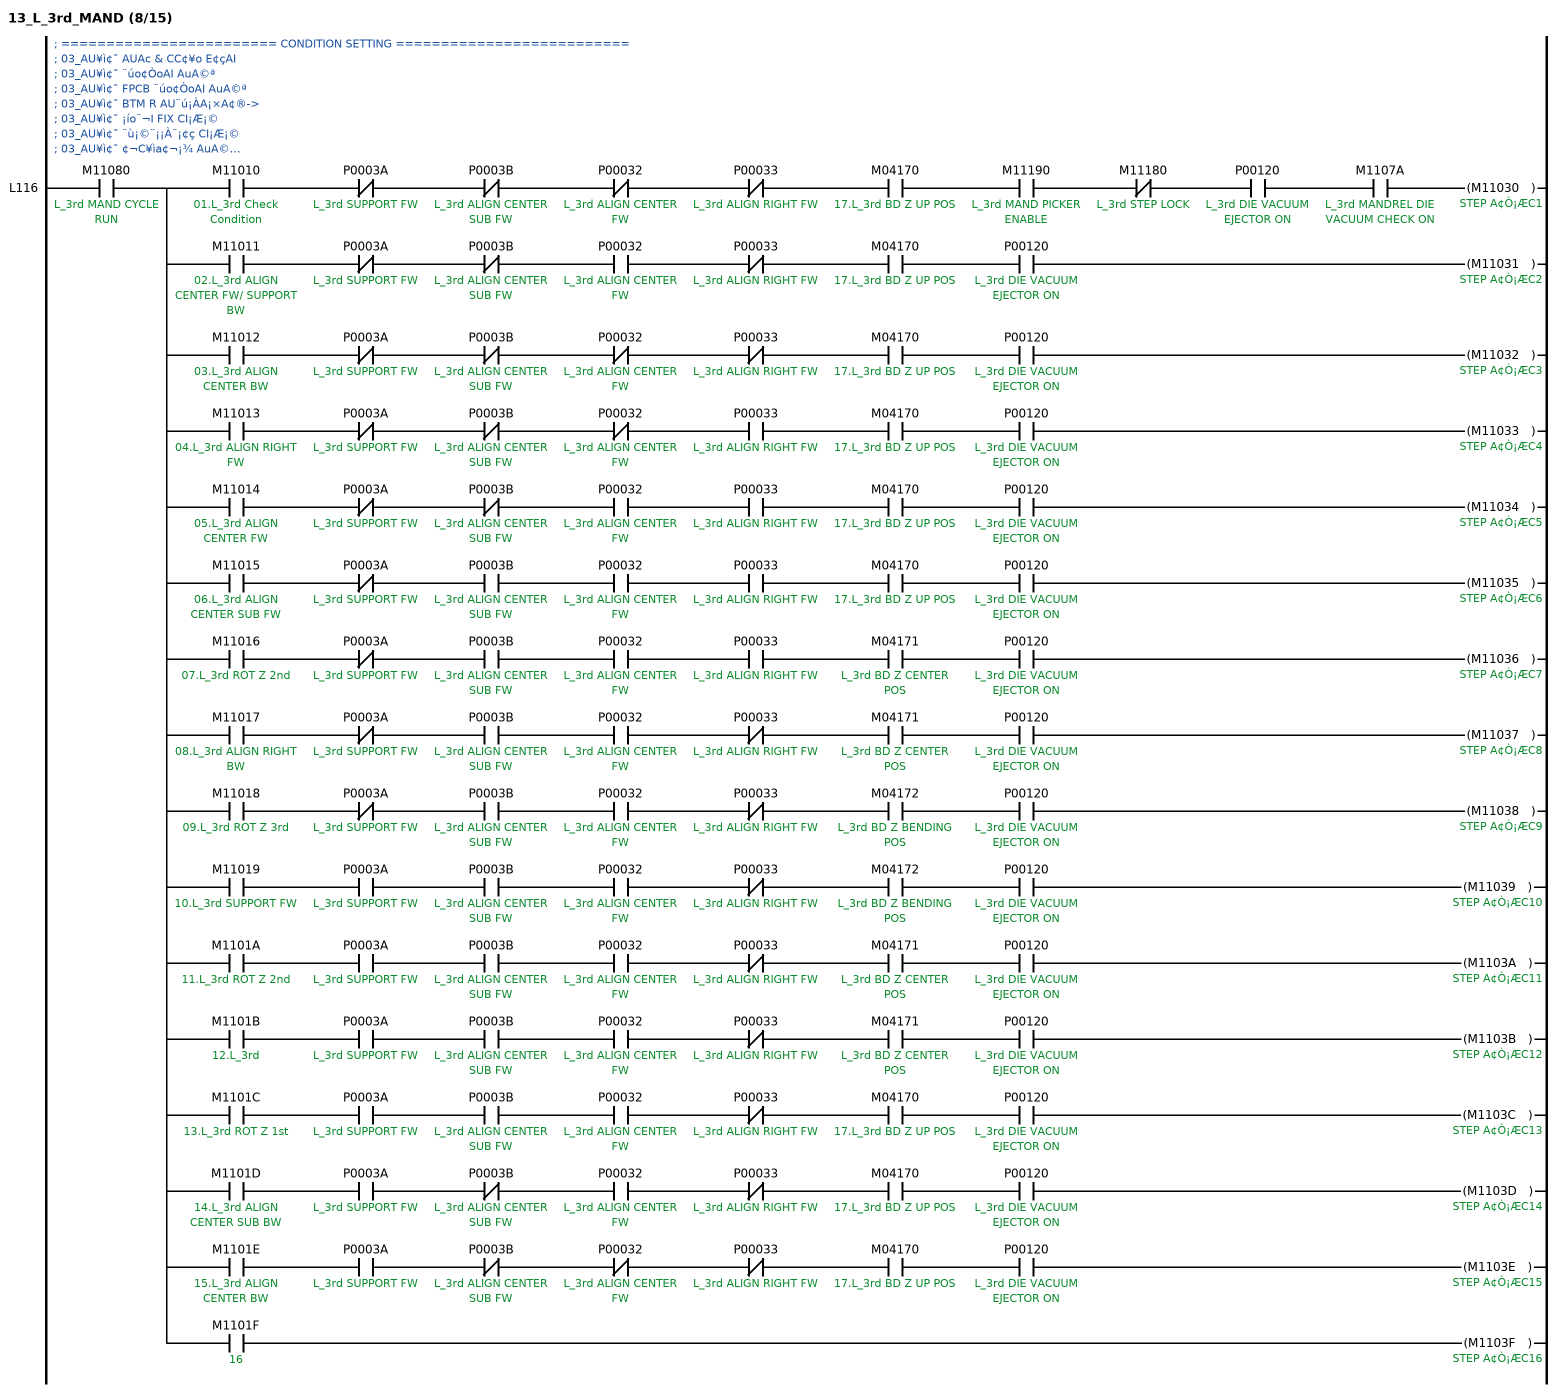
// ======================== CONDITION SETTING ==========================
; L116
LOAD      M11080	// L_3rd MAND CYCLE RUN
MPUSH
AND       M11010	// 01.L_3rd Check Condition
AND NOT   P0003A	// L_3rd SUPPORT FW
AND NOT   P0003B	// L_3rd ALIGN CENTER SUB FW
AND NOT   P00032	// L_3rd ALIGN CENTER FW
AND NOT   P00033	// L_3rd ALIGN RIGHT FW
AND       M04170	// 17.L_3rd BD Z UP POS
AND       M11190	// L_3rd MAND PICKER ENABLE
AND NOT   M11180	// L_3rd STEP LOCK
AND       P00120	// L_3rd DIE VACUUM EJECTOR ON
AND       M1107A	// L_3rd MANDREL DIE VACUUM CHECK ON
OUT       M11030	// STEP A¢Ò¡ÆC1
MLOAD
AND       M11011	// 02.L_3rd ALIGN CENTER FW/ SUPPORT BW
AND NOT   P0003A	// L_3rd SUPPORT FW
AND NOT   P0003B	// L_3rd ALIGN CENTER SUB FW
AND       P00032	// L_3rd ALIGN CENTER FW
AND NOT   P00033	// L_3rd ALIGN RIGHT FW
AND       M04170	// 17.L_3rd BD Z UP POS
AND       P00120	// L_3rd DIE VACUUM EJECTOR ON
OUT       M11031	// STEP A¢Ò¡ÆC2
MLOAD
AND       M11012	// 03.L_3rd ALIGN CENTER BW
AND NOT   P0003A	// L_3rd SUPPORT FW
AND NOT   P0003B	// L_3rd ALIGN CENTER SUB FW
AND NOT   P00032	// L_3rd ALIGN CENTER FW
AND NOT   P00033	// L_3rd ALIGN RIGHT FW
AND       M04170	// 17.L_3rd BD Z UP POS
AND       P00120	// L_3rd DIE VACUUM EJECTOR ON
OUT       M11032	// STEP A¢Ò¡ÆC3
MLOAD
AND       M11013	// 04.L_3rd ALIGN RIGHT FW
AND NOT   P0003A	// L_3rd SUPPORT FW
AND NOT   P0003B	// L_3rd ALIGN CENTER SUB FW
AND NOT   P00032	// L_3rd ALIGN CENTER FW
AND       P00033	// L_3rd ALIGN RIGHT FW
AND       M04170	// 17.L_3rd BD Z UP POS
AND       P00120	// L_3rd DIE VACUUM EJECTOR ON
OUT       M11033	// STEP A¢Ò¡ÆC4
MLOAD
AND       M11014	// 05.L_3rd ALIGN CENTER FW
AND NOT   P0003A	// L_3rd SUPPORT FW
AND NOT   P0003B	// L_3rd ALIGN CENTER SUB FW
AND       P00032	// L_3rd ALIGN CENTER FW
AND       P00033	// L_3rd ALIGN RIGHT FW
AND       M04170	// 17.L_3rd BD Z UP POS
AND       P00120	// L_3rd DIE VACUUM EJECTOR ON
OUT       M11034	// STEP A¢Ò¡ÆC5
MLOAD
AND       M11015	// 06.L_3rd ALIGN CENTER SUB FW
AND NOT   P0003A	// L_3rd SUPPORT FW
AND       P0003B	// L_3rd ALIGN CENTER SUB FW
AND       P00032	// L_3rd ALIGN CENTER FW
AND       P00033	// L_3rd ALIGN RIGHT FW
AND       M04170	// 17.L_3rd BD Z UP POS
AND       P00120	// L_3rd DIE VACUUM EJECTOR ON
OUT       M11035	// STEP A¢Ò¡ÆC6
MLOAD
AND       M11016	// 07.L_3rd ROT Z 2nd
AND NOT   P0003A	// L_3rd SUPPORT FW
AND       P0003B	// L_3rd ALIGN CENTER SUB FW
AND       P00032	// L_3rd ALIGN CENTER FW
AND       P00033	// L_3rd ALIGN RIGHT FW
AND       M04171	// L_3rd BD Z CENTER POS
AND       P00120	// L_3rd DIE VACUUM EJECTOR ON
OUT       M11036	// STEP A¢Ò¡ÆC7
MLOAD
AND       M11017	// 08.L_3rd ALIGN RIGHT BW
AND NOT   P0003A	// L_3rd SUPPORT FW
AND       P0003B	// L_3rd ALIGN CENTER SUB FW
AND       P00032	// L_3rd ALIGN CENTER FW
AND NOT   P00033	// L_3rd ALIGN RIGHT FW
AND       M04171	// L_3rd BD Z CENTER POS
AND       P00120	// L_3rd DIE VACUUM EJECTOR ON
OUT       M11037	// STEP A¢Ò¡ÆC8
MLOAD
AND       M11018	// 09.L_3rd ROT Z 3rd
AND NOT   P0003A	// L_3rd SUPPORT FW
AND       P0003B	// L_3rd ALIGN CENTER SUB FW
AND       P00032	// L_3rd ALIGN CENTER FW
AND NOT   P00033	// L_3rd ALIGN RIGHT FW
AND       M04172	// L_3rd BD Z BENDING POS
AND       P00120	// L_3rd DIE VACUUM EJECTOR ON
OUT       M11038	// STEP A¢Ò¡ÆC9
MLOAD
AND       M11019	// 10.L_3rd SUPPORT FW
AND       P0003A	// L_3rd SUPPORT FW
AND       P0003B	// L_3rd ALIGN CENTER SUB FW
AND       P00032	// L_3rd ALIGN CENTER FW
AND NOT   P00033	// L_3rd ALIGN RIGHT FW
AND       M04172	// L_3rd BD Z BENDING POS
AND       P00120	// L_3rd DIE VACUUM EJECTOR ON
OUT       M11039	// STEP A¢Ò¡ÆC10
MLOAD
AND       M1101A	// 11.L_3rd ROT Z 2nd
AND       P0003A	// L_3rd SUPPORT FW
AND       P0003B	// L_3rd ALIGN CENTER SUB FW
AND       P00032	// L_3rd ALIGN CENTER FW
AND NOT   P00033	// L_3rd ALIGN RIGHT FW
AND       M04171	// L_3rd BD Z CENTER POS
AND       P00120	// L_3rd DIE VACUUM EJECTOR ON
OUT       M1103A	// STEP A¢Ò¡ÆC11
MLOAD
AND       M1101B	// 12.L_3rd 
AND       P0003A	// L_3rd SUPPORT FW
AND       P0003B	// L_3rd ALIGN CENTER SUB FW
AND       P00032	// L_3rd ALIGN CENTER FW
AND NOT   P00033	// L_3rd ALIGN RIGHT FW
AND       M04171	// L_3rd BD Z CENTER POS
AND       P00120	// L_3rd DIE VACUUM EJECTOR ON
OUT       M1103B	// STEP A¢Ò¡ÆC12
MLOAD
AND       M1101C	// 13.L_3rd ROT Z 1st
AND       P0003A	// L_3rd SUPPORT FW
AND       P0003B	// L_3rd ALIGN CENTER SUB FW
AND       P00032	// L_3rd ALIGN CENTER FW
AND NOT   P00033	// L_3rd ALIGN RIGHT FW
AND       M04170	// 17.L_3rd BD Z UP POS
AND       P00120	// L_3rd DIE VACUUM EJECTOR ON
OUT       M1103C	// STEP A¢Ò¡ÆC13
MLOAD
AND       M1101D	// 14.L_3rd ALIGN CENTER SUB BW
AND       P0003A	// L_3rd SUPPORT FW
AND NOT   P0003B	// L_3rd ALIGN CENTER SUB FW
AND       P00032	// L_3rd ALIGN CENTER FW
AND NOT   P00033	// L_3rd ALIGN RIGHT FW
AND       M04170	// 17.L_3rd BD Z UP POS
AND       P00120	// L_3rd DIE VACUUM EJECTOR ON
OUT       M1103D	// STEP A¢Ò¡ÆC14
MLOAD
AND       M1101E	// 15.L_3rd ALIGN CENTER BW
AND       P0003A	// L_3rd SUPPORT FW
AND NOT   P0003B	// L_3rd ALIGN CENTER SUB FW
AND NOT   P00032	// L_3rd ALIGN CENTER FW
AND NOT   P00033	// L_3rd ALIGN RIGHT FW
AND       M04170	// 17.L_3rd BD Z UP POS
AND       P00120	// L_3rd DIE VACUUM EJECTOR ON
OUT       M1103E	// STEP A¢Ò¡ÆC15
MPOP
AND       M1101F	// 16
OUT       M1103F	// STEP A¢Ò¡ÆC16
// output comment: 03_AU¥ì¢¯ AUAc & CC¢¥o E¢çAI
// output comment: 03_AU¥ì¢¯ ¨úo¢ÒoAI AuA©ª
// output comment: 03_AU¥ì¢¯ FPCB ¨úo¢ÒoAI AuA©ª
// output comment: 03_AU¥ì¢¯ BTM R AU¨ú¡ÀA¡×A¢®->
// output comment: 03_AU¥ì¢¯ ¡ío¨¬I FIX CI¡Æ¡©
// output comment: 03_AU¥ì¢¯ ¨ù¡©¨¡¡À¨¡¢ç CI¡Æ¡©
// output comment: 03_AU¥ì¢¯ ¢¬C¥ìa¢¬¡¾ AuA©ª
// output comment: 03_AU¥ì¢¯ ¢¬C¥ìa¢¬¡¾ E¢¬Au
// output comment: 03_AU¥ì¢¯ ¢¬C¥ìa¢¬¡¾ ¨¬©ö¡¾I
// output comment: 03_AU¥ì¢¯ ¢¬C¥ìa¢¬¡¾ EAA©ª
// output comment: 03_AU¥ì¢¯ ¡ío¨¬I ¡¤¢®A¢® CI¡Æ¡©
// output comment: 03_AU¥ì¢¯ Y ¨ö¨¬¨¡CA¡¤ IN -> ¢¬a¥ìa¢¬¡¾ ¢¥e¡¾a->
// output comment: 03_AU¥ì¢¯ ¨ö¨¬¨¡CA¡¤ AuA©ª
// output comment: 03_AU¥ì¢¯ Y ¨ö¨¬¨¡CA¡¤ A¡×A¢®
// output comment: 03_AU¥ì¢¯ Y ¨ö¨¬¨¡CA¡¤ IN->
// output comment: 03_AU¥ì¢¯ ¨ö¨¬¨¡CA¡¤ EAA©ª ,¡ío¨¬I ¡¤¢®A¢® ¡ío¨öA

